Yaskawa INFORM job: A_ROOF_UPPER_0614_2_PAINT_9.JBI

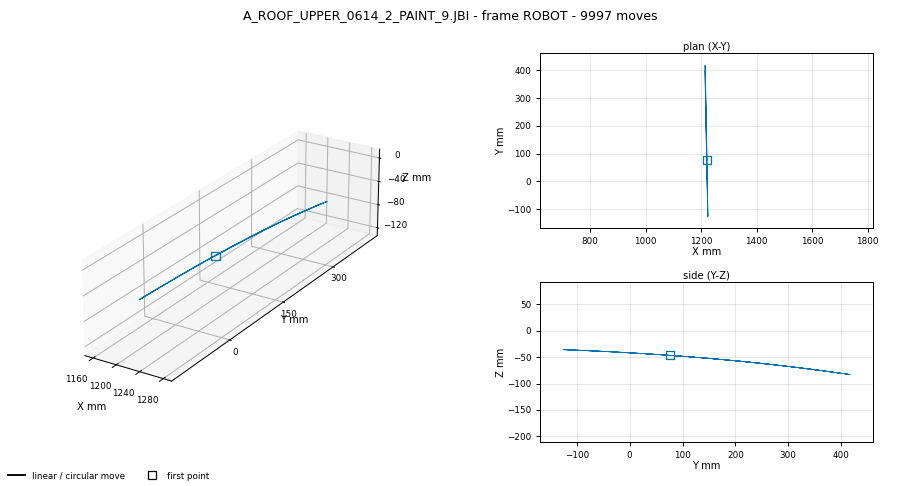
[picture p0: tool path of A_ROOF_UPPER_0614_2_PAINT_9.JBI in frame ROBOT, 9997 of 9997 moves have a stored position in this frame; points joined in program order, loops and branches not executed]
/JOB
//NAME A_ROOF_UPPER_0614_2_PAINT9
//POS
///NPOS 9997,0,0,0,0,0
///TOOL 1
///USER 0
///POSTYPE ROBOT
///RECTAN
///RCONF 1,0,0,0,0,0,0,0,0,0,0,0,0,0,0,0,0,0,0,0,0,0,0,0
C00000=1221.540,75.993,-46.507,-178.760,5.552,148.601
C00001=1221.535,76.242,-46.525,-178.757,5.552,148.601
C00002=1221.530,76.492,-46.542,-178.755,5.553,148.600
C00003=1221.525,76.741,-46.560,-178.753,5.554,148.600
C00004=1221.520,76.990,-46.578,-178.750,5.554,148.599
C00005=1221.515,77.240,-46.595,-178.747,5.555,148.598
C00006=1221.510,77.489,-46.613,-178.745,5.557,148.598
C00007=1221.505,77.738,-46.631,-178.742,5.557,148.597
C00008=1221.501,77.988,-46.648,-178.739,5.558,148.596
C00009=1221.496,78.237,-46.666,-178.737,5.559,148.596
C00010=1221.491,78.486,-46.684,-178.735,5.559,148.595
C00011=1221.486,78.735,-46.702,-178.732,5.560,148.595
C00012=1221.481,78.985,-46.719,-178.729,5.560,148.594
C00013=1221.476,79.234,-46.737,-178.727,5.561,148.594
C00014=1221.471,79.484,-46.755,-178.725,5.562,148.593
C00015=1221.466,79.733,-46.773,-178.722,5.563,148.592
C00016=1221.462,79.982,-46.790,-178.719,5.564,148.592
C00017=1221.457,80.231,-46.808,-178.717,5.565,148.591
C00018=1221.452,80.481,-46.826,-178.714,5.566,148.591
C00019=1221.448,80.730,-46.844,-178.711,5.566,148.590
C00020=1221.443,80.980,-46.862,-178.709,5.567,148.589
C00021=1221.437,81.249,-46.881,-178.707,5.568,148.589
C00022=1221.432,81.516,-46.900,-178.703,5.569,148.588
C00023=1221.427,81.784,-46.919,-178.701,5.570,148.588
C00024=1221.421,82.053,-46.939,-178.698,5.570,148.587
C00025=1221.416,82.302,-46.956,-178.696,5.571,148.586
C00026=1221.411,82.552,-46.974,-178.693,5.571,148.586
C00027=1221.407,82.801,-46.992,-178.690,5.573,148.585
C00028=1221.402,83.051,-47.010,-178.688,5.574,148.585
C00029=1221.397,83.300,-47.028,-178.685,5.574,148.584
C00030=1221.392,83.549,-47.046,-178.682,5.575,148.583
C00031=1221.387,83.798,-47.064,-178.680,5.576,148.583
C00032=1221.382,84.047,-47.082,-178.678,5.576,148.582
C00033=1221.378,84.296,-47.100,-178.675,5.577,148.581
C00034=1221.373,84.546,-47.118,-178.672,5.579,148.581
C00035=1221.368,84.796,-47.136,-178.670,5.579,148.580
C00036=1221.363,85.045,-47.154,-178.667,5.580,148.580
C00037=1221.358,85.294,-47.172,-178.664,5.581,148.579
C00038=1221.353,85.544,-47.190,-178.662,5.582,148.579
C00039=1221.348,85.793,-47.208,-178.660,5.582,148.578
C00040=1221.343,86.042,-47.226,-178.657,5.583,148.577
C00041=1221.339,86.291,-47.244,-178.654,5.584,148.577
C00042=1221.334,86.541,-47.262,-178.652,5.585,148.576
C00043=1221.329,86.790,-47.280,-178.649,5.586,148.576
C00044=1221.324,87.040,-47.298,-178.647,5.587,148.575
C00045=1221.319,87.289,-47.316,-178.644,5.587,148.575
C00046=1221.314,87.538,-47.334,-178.642,5.588,148.574
C00047=1221.309,87.787,-47.353,-178.639,5.588,148.573
C00048=1221.305,88.037,-47.371,-178.636,5.590,148.573
C00049=1221.300,88.286,-47.389,-178.634,5.591,148.572
C00050=1221.295,88.535,-47.407,-178.631,5.591,148.572
C00051=1221.290,88.784,-47.425,-178.629,5.592,148.571
C00052=1221.285,89.033,-47.443,-178.626,5.593,148.570
C00053=1221.281,89.283,-47.462,-178.624,5.593,148.570
C00054=1221.275,89.533,-47.480,-178.621,5.595,148.569
C00055=1221.270,89.782,-47.498,-178.618,5.596,148.569
C00056=1221.266,90.031,-47.516,-178.616,5.596,148.568
C00057=1221.261,90.279,-47.535,-178.614,5.597,148.568
C00058=1221.257,90.529,-47.553,-178.611,5.598,148.567
C00059=1221.252,90.779,-47.571,-178.608,5.599,148.566
C00060=1221.246,91.028,-47.590,-178.605,5.600,148.566
C00061=1221.241,91.277,-47.608,-178.603,5.601,148.565
C00062=1221.237,91.527,-47.626,-178.601,5.601,148.565
C00063=1221.232,91.776,-47.645,-178.598,5.602,148.564
C00064=1221.227,92.025,-47.663,-178.596,5.603,148.564
C00065=1221.222,92.274,-47.681,-178.593,5.604,148.563
C00066=1221.217,92.524,-47.700,-178.590,5.605,148.562
C00067=1221.212,92.773,-47.718,-178.588,5.606,148.562
C00068=1221.208,93.022,-47.736,-178.585,5.607,148.561
C00069=1221.203,93.271,-47.754,-178.583,5.607,148.561
C00070=1221.198,93.521,-47.773,-178.580,5.608,148.560
C00071=1221.193,93.770,-47.792,-178.577,5.610,148.560
C00072=1221.188,94.019,-47.810,-178.575,5.610,148.559
C00073=1221.183,94.268,-47.828,-178.573,5.611,148.558
C00074=1221.178,94.518,-47.847,-178.570,5.612,148.558
C00075=1221.174,94.767,-47.866,-178.567,5.612,148.557
C00076=1221.169,95.016,-47.884,-178.565,5.614,148.557
C00077=1221.165,95.266,-47.902,-178.562,5.615,148.556
C00078=1221.159,95.515,-47.921,-178.559,5.615,148.555
C00079=1221.154,95.764,-47.939,-178.557,5.616,148.555
C00080=1221.149,96.013,-47.957,-178.555,5.617,148.554
C00081=1221.145,96.263,-47.977,-178.551,5.618,148.554
C00082=1221.140,96.512,-47.995,-178.549,5.619,148.553
C00083=1221.135,96.761,-48.013,-178.547,5.620,148.553
C00084=1221.131,97.010,-48.032,-178.544,5.620,148.552
C00085=1221.125,97.260,-48.050,-178.542,5.621,148.552
C00086=1221.121,97.508,-48.069,-178.539,5.623,148.551
C00087=1221.116,97.758,-48.087,-178.537,5.624,148.551
C00088=1221.111,98.008,-48.106,-178.534,5.624,148.550
C00089=1221.106,98.256,-48.125,-178.531,5.625,148.549
C00090=1221.102,98.506,-48.143,-178.529,5.626,148.549
C00091=1221.096,98.755,-48.162,-178.526,5.627,148.548
C00092=1221.091,99.004,-48.180,-178.523,5.628,148.548
C00093=1221.087,99.254,-48.200,-178.521,5.629,148.547
C00094=1221.082,99.503,-48.218,-178.519,5.629,148.546
C00095=1221.078,99.752,-48.237,-178.516,5.631,148.546
C00096=1221.072,100.002,-48.256,-178.513,5.632,148.545
C00097=1221.068,100.250,-48.274,-178.511,5.632,148.545
C00098=1221.062,100.500,-48.293,-178.508,5.633,148.544
C00099=1221.058,100.749,-48.312,-178.506,5.634,148.544
C00100=1221.053,100.998,-48.330,-178.503,5.635,148.543
C00101=1221.048,101.248,-48.350,-178.501,5.636,148.543
C00102=1221.043,101.497,-48.368,-178.498,5.637,148.542
C00103=1221.039,101.747,-48.387,-178.496,5.638,148.541
C00104=1221.034,101.996,-48.405,-178.493,5.639,148.541
C00105=1221.028,102.245,-48.425,-178.490,5.640,148.540
C00106=1221.024,102.494,-48.444,-178.488,5.641,148.540
C00107=1221.019,102.743,-48.462,-178.485,5.641,148.539
C00108=1221.015,102.993,-48.481,-178.482,5.643,148.539
C00109=1221.010,103.242,-48.499,-178.480,5.644,148.538
C00110=1221.005,103.491,-48.519,-178.478,5.644,148.538
C00111=1221.000,103.740,-48.538,-178.475,5.645,148.537
C00112=1220.995,103.989,-48.556,-178.472,5.647,148.537
C00113=1220.991,104.239,-48.575,-178.470,5.647,148.536
C00114=1220.985,104.487,-48.594,-178.467,5.648,148.535
C00115=1220.981,104.737,-48.613,-178.465,5.649,148.535
C00116=1220.976,104.986,-48.632,-178.462,5.650,148.534
C00117=1220.972,105.235,-48.651,-178.460,5.651,148.534
C00118=1220.966,105.485,-48.670,-178.457,5.652,148.533
C00119=1220.961,105.735,-48.689,-178.454,5.653,148.532
C00120=1220.957,105.983,-48.708,-178.452,5.654,148.532
C00121=1220.952,106.233,-48.727,-178.449,5.655,148.531
C00122=1220.947,106.482,-48.746,-178.447,5.656,148.531
C00123=1220.942,106.731,-48.765,-178.444,5.657,148.530
C00124=1220.938,106.980,-48.784,-178.441,5.658,148.530
C00125=1220.932,107.249,-48.804,-178.439,5.659,148.529
C00126=1220.927,107.517,-48.825,-178.436,5.660,148.529
C00127=1220.921,107.785,-48.846,-178.433,5.661,148.528
C00128=1220.916,108.054,-48.866,-178.431,5.662,148.527
C00129=1220.912,108.303,-48.885,-178.428,5.663,148.527
C00130=1220.907,108.553,-48.905,-178.425,5.664,148.526
C00131=1220.903,108.802,-48.924,-178.423,5.665,148.526
C00132=1220.898,109.051,-48.943,-178.421,5.666,148.525
C00133=1220.892,109.301,-48.962,-178.417,5.667,148.525
C00134=1220.888,109.549,-48.981,-178.415,5.668,148.524
C00135=1220.883,109.799,-49.000,-178.413,5.669,148.524
C00136=1220.878,110.048,-49.020,-178.409,5.670,148.523
C00137=1220.874,110.297,-49.039,-178.407,5.671,148.523
C00138=1220.868,110.546,-49.058,-178.405,5.672,148.522
C00139=1220.864,110.796,-49.078,-178.403,5.673,148.522
C00140=1220.859,111.044,-49.096,-178.399,5.674,148.521
C00141=1220.854,111.294,-49.115,-178.397,5.675,148.520
C00142=1220.849,111.543,-49.134,-178.395,5.676,148.520
C00143=1220.845,111.792,-49.154,-178.392,5.677,148.519
C00144=1220.840,112.042,-49.173,-178.389,5.678,148.519
C00145=1220.835,112.291,-49.192,-178.387,5.679,148.518
C00146=1220.831,112.540,-49.212,-178.385,5.679,148.518
C00147=1220.825,112.789,-49.231,-178.381,5.681,148.517
C00148=1220.821,113.039,-49.250,-178.379,5.682,148.516
C00149=1220.815,113.287,-49.270,-178.377,5.682,148.516
C00150=1220.811,113.537,-49.289,-178.374,5.684,148.515
C00151=1220.806,113.786,-49.309,-178.371,5.685,148.515
C00152=1220.801,114.035,-49.328,-178.369,5.686,148.514
C00153=1220.796,114.285,-49.347,-178.367,5.686,148.514
C00154=1220.792,114.533,-49.366,-178.364,5.688,148.513
C00155=1220.787,114.783,-49.386,-178.361,5.689,148.513
C00156=1220.782,115.032,-49.405,-178.359,5.689,148.512
C00157=1220.777,115.281,-49.425,-178.356,5.691,148.512
C00158=1220.773,115.530,-49.444,-178.354,5.692,148.511
C00159=1220.768,115.780,-49.463,-178.351,5.692,148.511
C00160=1220.763,116.029,-49.483,-178.348,5.694,148.510
C00161=1220.758,116.278,-49.503,-178.346,5.695,148.510
C00162=1220.753,116.527,-49.522,-178.343,5.696,148.509
C00163=1220.748,116.776,-49.542,-178.340,5.697,148.509
C00164=1220.744,117.026,-49.561,-178.338,5.698,148.508
C00165=1220.739,117.274,-49.580,-178.336,5.699,148.507
C00166=1220.734,117.524,-49.600,-178.332,5.700,148.507
C00167=1220.729,117.774,-49.620,-178.330,5.701,148.506
C00168=1220.724,118.022,-49.639,-178.328,5.702,148.506
C00169=1220.720,118.271,-49.659,-178.325,5.704,148.505
C00170=1220.716,118.521,-49.678,-178.322,5.704,148.505
C00171=1220.710,118.769,-49.698,-178.320,5.705,148.504
C00172=1220.706,119.019,-49.717,-178.317,5.707,148.504
C00173=1220.701,119.269,-49.737,-178.315,5.708,148.503
C00174=1220.696,119.517,-49.757,-178.312,5.708,148.503
C00175=1220.691,119.766,-49.777,-178.309,5.710,148.502
C00176=1220.686,120.016,-49.796,-178.307,5.711,148.502
C00177=1220.682,120.266,-49.816,-178.304,5.711,148.501
C00178=1220.677,120.514,-49.836,-178.302,5.713,148.501
C00179=1220.672,120.763,-49.856,-178.299,5.714,148.500
C00180=1220.668,121.013,-49.875,-178.297,5.715,148.500
C00181=1220.662,121.261,-49.894,-178.294,5.716,148.499
C00182=1220.658,121.510,-49.914,-178.292,5.717,148.499
C00183=1220.653,121.760,-49.934,-178.289,5.718,148.498
C00184=1220.649,122.010,-49.954,-178.286,5.720,148.498
C00185=1220.643,122.258,-49.974,-178.284,5.720,148.497
C00186=1220.639,122.507,-49.993,-178.282,5.721,148.496
C00187=1220.634,122.757,-50.013,-178.279,5.723,148.496
C00188=1220.630,123.006,-50.033,-178.276,5.723,148.495
C00189=1220.624,123.255,-50.053,-178.274,5.724,148.495
C00190=1220.619,123.504,-50.072,-178.271,5.726,148.494
C00191=1220.615,123.753,-50.093,-178.269,5.727,148.494
C00192=1220.610,124.003,-50.112,-178.266,5.727,148.493
C00193=1220.605,124.251,-50.132,-178.263,5.729,148.493
C00194=1220.601,124.501,-50.152,-178.261,5.730,148.492
C00195=1220.596,124.750,-50.172,-178.258,5.731,148.492
C00196=1220.591,124.999,-50.192,-178.255,5.732,148.491
C00197=1220.586,125.248,-50.211,-178.253,5.733,148.491
C00198=1220.582,125.497,-50.232,-178.250,5.734,148.490
C00199=1220.577,125.747,-50.251,-178.248,5.735,148.490
C00200=1220.572,125.996,-50.272,-178.245,5.736,148.489
C00201=1220.568,126.245,-50.291,-178.243,5.738,148.489
C00202=1220.562,126.494,-50.312,-178.240,5.738,148.488
C00203=1220.557,126.743,-50.332,-178.238,5.739,148.488
C00204=1220.553,126.992,-50.352,-178.235,5.741,148.487
C00205=1220.548,127.242,-50.372,-178.233,5.742,148.487
C00206=1220.543,127.491,-50.392,-178.230,5.743,148.486
C00207=1220.539,127.740,-50.412,-178.227,5.744,148.486
C00208=1220.534,127.989,-50.432,-178.225,5.745,148.485
C00209=1220.529,128.238,-50.451,-178.222,5.747,148.485
C00210=1220.525,128.487,-50.472,-178.220,5.747,148.484
C00211=1220.520,128.737,-50.491,-178.217,5.749,148.484
C00212=1220.515,128.986,-50.512,-178.214,5.750,148.483
C00213=1220.510,129.235,-50.532,-178.212,5.751,148.482
C00214=1220.505,129.484,-50.552,-178.209,5.752,148.482
C00215=1220.500,129.733,-50.572,-178.207,5.753,148.481
C00216=1220.496,129.982,-50.592,-178.205,5.754,148.481
C00217=1220.491,130.231,-50.612,-178.202,5.755,148.480
C00218=1220.487,130.480,-50.633,-178.199,5.756,148.480
C00219=1220.481,130.730,-50.653,-178.196,5.758,148.479
C00220=1220.477,130.979,-50.673,-178.194,5.759,148.479
C00221=1220.472,131.228,-50.694,-178.192,5.759,148.478
C00222=1220.467,131.477,-50.713,-178.189,5.761,148.478
C00223=1220.463,131.726,-50.734,-178.186,5.762,148.477
C00224=1220.457,131.975,-50.754,-178.184,5.764,148.477
C00225=1220.453,132.225,-50.774,-178.181,5.764,148.476
C00226=1220.448,132.473,-50.794,-178.178,5.766,148.476
C00227=1220.444,132.722,-50.815,-178.176,5.767,148.475
C00228=1220.438,132.972,-50.835,-178.174,5.768,148.475
C00229=1220.434,133.240,-50.857,-178.170,5.769,148.474
C00230=1220.428,133.509,-50.879,-178.168,5.771,148.474
C00231=1220.423,133.778,-50.901,-178.165,5.772,148.473
C00232=1220.418,134.047,-50.922,-178.162,5.773,148.473
C00233=1220.413,134.296,-50.943,-178.160,5.774,148.472
C00234=1220.408,134.544,-50.963,-178.157,5.776,148.472
C00235=1220.404,134.793,-50.984,-178.155,5.776,148.471
C00236=1220.399,135.042,-51.004,-178.152,5.777,148.471
C00237=1220.394,135.292,-51.024,-178.149,5.779,148.470
C00238=1220.389,135.541,-51.045,-178.147,5.780,148.470
C00239=1220.385,135.790,-51.065,-178.144,5.781,148.469
C00240=1220.380,136.039,-51.086,-178.142,5.782,148.469
C00241=1220.375,136.288,-51.107,-178.139,5.784,148.468
C00242=1220.371,136.537,-51.127,-178.137,5.785,148.468
C00243=1220.366,136.787,-51.148,-178.134,5.785,148.467
C00244=1220.361,137.036,-51.167,-178.131,5.787,148.467
C00245=1220.357,137.285,-51.188,-178.129,5.788,148.466
C00246=1220.351,137.534,-51.209,-178.126,5.790,148.466
C00247=1220.347,137.783,-51.229,-178.124,5.791,148.465
C00248=1220.343,138.032,-51.250,-178.121,5.792,148.465
C00249=1220.337,138.282,-51.271,-178.119,5.793,148.464
C00250=1220.333,138.530,-51.291,-178.116,5.794,148.464
C00251=1220.328,138.780,-51.312,-178.113,5.795,148.463
C00252=1220.323,139.029,-51.332,-178.111,5.796,148.463
C00253=1220.319,139.278,-51.353,-178.108,5.798,148.462
C00254=1220.314,139.527,-51.374,-178.106,5.799,148.462
C00255=1220.309,139.776,-51.394,-178.103,5.800,148.461
C00256=1220.304,140.025,-51.415,-178.101,5.801,148.461
C00257=1220.300,140.274,-51.435,-178.098,5.803,148.460
C00258=1220.294,140.523,-51.456,-178.095,5.804,148.460
C00259=1220.290,140.772,-51.477,-178.092,5.805,148.459
C00260=1220.286,141.021,-51.497,-178.090,5.806,148.459
C00261=1220.280,141.270,-51.518,-178.088,5.808,148.459
C00262=1220.276,141.519,-51.538,-178.085,5.809,148.458
C00263=1220.271,141.769,-51.559,-178.083,5.810,148.458
C00264=1220.266,142.018,-51.580,-178.080,5.811,148.457
C00265=1220.262,142.268,-51.601,-178.078,5.812,148.457
C00266=1220.257,142.517,-51.621,-178.074,5.813,148.456
C00267=1220.252,142.766,-51.642,-178.072,5.814,148.456
C00268=1220.248,143.014,-51.663,-178.070,5.816,148.455
C00269=1220.243,143.263,-51.684,-178.067,5.817,148.454
C00270=1220.238,143.512,-51.705,-178.064,5.819,148.454
C00271=1220.233,143.762,-51.726,-178.062,5.819,148.453
C00272=1220.229,144.011,-51.746,-178.059,5.821,148.453
C00273=1220.224,144.260,-51.767,-178.057,5.822,148.453
C00274=1220.220,144.508,-51.788,-178.054,5.824,148.452
C00275=1220.215,144.758,-51.810,-178.052,5.825,148.452
C00276=1220.210,145.007,-51.830,-178.049,5.826,148.451
C00277=1220.205,145.256,-51.851,-178.046,5.827,148.451
C00278=1220.200,145.506,-51.872,-178.044,5.829,148.450
C00279=1220.196,145.754,-51.893,-178.041,5.829,148.450
C00280=1220.191,146.003,-51.914,-178.039,5.831,148.449
C00281=1220.186,146.252,-51.934,-178.036,5.832,148.449
C00282=1220.181,146.501,-51.955,-178.033,5.834,148.448
C00283=1220.177,146.751,-51.977,-178.031,5.835,148.448
C00284=1220.173,147.000,-51.998,-178.028,5.836,148.447
C00285=1220.167,147.249,-52.019,-178.026,5.837,148.447
C00286=1220.162,147.498,-52.040,-178.023,5.839,148.447
C00287=1220.158,147.746,-52.061,-178.021,5.840,148.446
C00288=1220.153,147.996,-52.082,-178.018,5.841,148.446
C00289=1220.148,148.245,-52.102,-178.015,5.842,148.445
C00290=1220.144,148.494,-52.124,-178.013,5.844,148.445
C00291=1220.139,148.743,-52.145,-178.011,5.845,148.444
C00292=1220.135,148.992,-52.165,-178.007,5.846,148.444
C00293=1220.130,149.241,-52.187,-178.005,5.847,148.443
C00294=1220.125,149.490,-52.208,-178.003,5.849,148.443
C00295=1220.121,149.740,-52.229,-178.000,5.850,148.442
C00296=1220.116,149.988,-52.250,-177.997,5.852,148.442
C00297=1220.111,150.238,-52.271,-177.995,5.852,148.441
C00298=1220.106,150.486,-52.293,-177.992,5.854,148.441
C00299=1220.101,150.735,-52.313,-177.990,5.855,148.440
C00300=1220.097,150.985,-52.336,-177.987,5.856,148.440
C00301=1220.092,151.234,-52.356,-177.985,5.857,148.439
C00302=1220.087,151.483,-52.377,-177.982,5.859,148.439
C00303=1220.083,151.731,-52.399,-177.979,5.860,148.438
C00304=1220.078,151.981,-52.420,-177.977,5.862,148.438
C00305=1220.073,152.230,-52.442,-177.975,5.863,148.438
C00306=1220.069,152.479,-52.462,-177.972,5.864,148.437
C00307=1220.064,152.728,-52.484,-177.969,5.866,148.437
C00308=1220.059,152.977,-52.505,-177.967,5.867,148.436
C00309=1220.054,153.226,-52.527,-177.964,5.868,148.436
C00310=1220.049,153.476,-52.548,-177.962,5.869,148.435
C00311=1220.045,153.724,-52.569,-177.958,5.871,148.435
C00312=1220.040,153.973,-52.590,-177.956,5.872,148.434
C00313=1220.036,154.222,-52.612,-177.954,5.874,148.434
C00314=1220.031,154.471,-52.633,-177.951,5.874,148.433
C00315=1220.026,154.720,-52.654,-177.948,5.876,148.433
C00316=1220.022,154.969,-52.676,-177.946,5.877,148.433
C00317=1220.017,155.219,-52.697,-177.943,5.879,148.432
C00318=1220.012,155.467,-52.718,-177.941,5.880,148.432
C00319=1220.007,155.716,-52.740,-177.938,5.881,148.431
C00320=1220.003,155.966,-52.761,-177.935,5.883,148.431
C00321=1219.998,156.215,-52.783,-177.933,5.884,148.430
C00322=1219.993,156.464,-52.804,-177.930,5.886,148.430
C00323=1219.989,156.713,-52.826,-177.928,5.886,148.429
C00324=1219.984,156.961,-52.847,-177.925,5.888,148.429
C00325=1219.979,157.211,-52.868,-177.923,5.889,148.428
C00326=1219.975,157.460,-52.890,-177.920,5.891,148.428
C00327=1219.970,157.709,-52.912,-177.917,5.892,148.427
C00328=1219.965,157.957,-52.934,-177.915,5.893,148.427
C00329=1219.960,158.207,-52.955,-177.912,5.895,148.427
C00330=1219.956,158.456,-52.977,-177.910,5.896,148.426
C00331=1219.951,158.705,-52.998,-177.907,5.898,148.426
C00332=1219.946,158.955,-53.020,-177.905,5.899,148.425
C00333=1219.942,159.223,-53.043,-177.902,5.900,148.425
C00334=1219.936,159.492,-53.066,-177.899,5.902,148.424
C00335=1219.931,159.761,-53.089,-177.896,5.903,148.424
C00336=1219.926,160.030,-53.113,-177.894,5.904,148.423
C00337=1219.921,160.279,-53.135,-177.891,5.906,148.423
C00338=1219.917,160.529,-53.156,-177.888,5.908,148.422
C00339=1219.912,160.777,-53.178,-177.886,5.909,148.422
C00340=1219.907,161.026,-53.200,-177.883,5.910,148.421
C00341=1219.903,161.275,-53.222,-177.881,5.911,148.421
C00342=1219.898,161.524,-53.243,-177.878,5.913,148.421
C00343=1219.893,161.773,-53.265,-177.876,5.915,148.420
C00344=1219.888,162.023,-53.286,-177.873,5.915,148.420
C00345=1219.884,162.271,-53.308,-177.870,5.917,148.419
C00346=1219.879,162.521,-53.330,-177.868,5.918,148.419
C00347=1219.874,162.769,-53.352,-177.865,5.920,148.418
C00348=1219.870,163.019,-53.374,-177.862,5.922,148.418
C00349=1219.865,163.267,-53.396,-177.860,5.923,148.418
C00350=1219.860,163.516,-53.417,-177.857,5.924,148.417
C00351=1219.856,163.765,-53.439,-177.855,5.925,148.417
C00352=1219.851,164.014,-53.461,-177.852,5.927,148.416
C00353=1219.847,164.263,-53.483,-177.850,5.929,148.416
C00354=1219.841,164.512,-53.505,-177.847,5.929,148.415
C00355=1219.837,164.761,-53.527,-177.844,5.931,148.415
C00356=1219.832,165.010,-53.549,-177.842,5.932,148.414
C00357=1219.828,165.259,-53.571,-177.840,5.934,148.414
C00358=1219.823,165.508,-53.593,-177.837,5.935,148.414
C00359=1219.818,165.757,-53.614,-177.834,5.936,148.413
C00360=1219.814,166.006,-53.637,-177.832,5.938,148.413
C00361=1219.809,166.255,-53.658,-177.829,5.939,148.412
C00362=1219.805,166.504,-53.680,-177.827,5.941,148.412
C00363=1219.799,166.753,-53.703,-177.824,5.942,148.411
C00364=1219.795,167.002,-53.725,-177.822,5.943,148.411
C00365=1219.790,167.251,-53.746,-177.819,5.945,148.410
C00366=1219.786,167.500,-53.768,-177.816,5.947,148.410
C00367=1219.781,167.749,-53.790,-177.814,5.948,148.410
C00368=1219.777,167.998,-53.812,-177.811,5.950,148.409
C00369=1219.771,168.247,-53.835,-177.809,5.950,148.409
C00370=1219.767,168.496,-53.857,-177.806,5.952,148.408
C00371=1219.762,168.745,-53.879,-177.803,5.954,148.408
C00372=1219.758,168.994,-53.901,-177.801,5.955,148.408
C00373=1219.753,169.243,-53.923,-177.798,5.956,148.407
C00374=1219.748,169.492,-53.945,-177.795,5.958,148.407
C00375=1219.744,169.742,-53.967,-177.793,5.959,148.406
C00376=1219.739,169.990,-53.990,-177.791,5.961,148.406
C00377=1219.735,170.239,-54.012,-177.787,5.963,148.405
C00378=1219.729,170.488,-54.034,-177.785,5.963,148.405
C00379=1219.725,170.737,-54.056,-177.783,5.965,148.405
C00380=1219.721,170.985,-54.078,-177.780,5.967,148.404
C00381=1219.716,171.235,-54.100,-177.778,5.968,148.404
C00382=1219.711,171.484,-54.123,-177.775,5.970,148.403
C00383=1219.706,171.733,-54.145,-177.773,5.971,148.403
C00384=1219.703,171.982,-54.168,-177.770,5.972,148.402
C00385=1219.697,172.231,-54.190,-177.767,5.974,148.402
C00386=1219.693,172.480,-54.212,-177.765,5.975,148.402
C00387=1219.688,172.729,-54.234,-177.762,5.977,148.401
C00388=1219.683,172.978,-54.257,-177.760,5.979,148.401
C00389=1219.678,173.226,-54.279,-177.757,5.980,148.400
C00390=1219.674,173.476,-54.301,-177.754,5.981,148.400
C00391=1219.669,173.725,-54.324,-177.752,5.983,148.399
C00392=1219.664,173.973,-54.346,-177.750,5.984,148.399
C00393=1219.660,174.223,-54.368,-177.747,5.986,148.399
C00394=1219.655,174.472,-54.391,-177.744,5.987,148.398
C00395=1219.651,174.720,-54.413,-177.742,5.988,148.398
C00396=1219.647,174.969,-54.436,-177.739,5.990,148.397
C00397=1219.641,175.218,-54.458,-177.736,5.992,148.397
C00398=1219.637,175.467,-54.480,-177.734,5.993,148.397
C00399=1219.632,175.716,-54.503,-177.731,5.994,148.396
C00400=1219.627,175.965,-54.525,-177.728,5.996,148.396
C00401=1219.623,176.214,-54.548,-177.726,5.998,148.395
C00402=1219.618,176.463,-54.570,-177.724,5.999,148.395
C00403=1219.614,176.711,-54.593,-177.721,6.001,148.395
C00404=1219.609,176.961,-54.615,-177.718,6.002,148.394
C00405=1219.605,177.210,-54.638,-177.716,6.003,148.394
C00406=1219.600,177.458,-54.660,-177.713,6.005,148.393
C00407=1219.595,177.707,-54.683,-177.711,6.007,148.393
C00408=1219.591,177.957,-54.705,-177.708,6.008,148.393
C00409=1219.586,178.205,-54.728,-177.705,6.009,148.392
C00410=1219.581,178.454,-54.750,-177.703,6.011,148.392
C00411=1219.577,178.703,-54.774,-177.701,6.012,148.391
C00412=1219.572,178.952,-54.795,-177.698,6.014,148.391
C00413=1219.567,179.201,-54.819,-177.695,6.016,148.391
C00414=1219.563,179.450,-54.841,-177.692,6.017,148.390
C00415=1219.557,179.699,-54.864,-177.690,6.018,148.390
C00416=1219.553,179.947,-54.886,-177.687,6.020,148.389
C00417=1219.548,180.197,-54.909,-177.685,6.022,148.389
C00418=1219.544,180.446,-54.932,-177.683,6.023,148.388
C00419=1219.539,180.694,-54.955,-177.679,6.025,148.388
C00420=1219.535,180.944,-54.977,-177.677,6.026,148.388
C00421=1219.530,181.193,-55.000,-177.674,6.028,148.387
C00422=1219.525,181.442,-55.024,-177.672,6.029,148.387
C00423=1219.521,181.690,-55.045,-177.669,6.031,148.386
C00424=1219.516,181.939,-55.069,-177.667,6.033,148.386
C00425=1219.512,182.188,-55.091,-177.664,6.034,148.385
C00426=1219.507,182.438,-55.114,-177.662,6.035,148.385
C00427=1219.502,182.686,-55.136,-177.659,6.037,148.385
C00428=1219.498,182.935,-55.160,-177.656,6.039,148.384
C00429=1219.493,183.184,-55.183,-177.654,6.040,148.384
C00430=1219.489,183.433,-55.205,-177.651,6.042,148.384
C00431=1219.483,183.681,-55.228,-177.648,6.043,148.383
C00432=1219.479,183.930,-55.251,-177.646,6.044,148.383
C00433=1219.475,184.179,-55.274,-177.644,6.046,148.382
C00434=1219.470,184.429,-55.297,-177.641,6.048,148.382
C00435=1219.466,184.678,-55.320,-177.638,6.050,148.382
C00436=1219.460,184.926,-55.343,-177.636,6.051,148.381
C00437=1219.455,185.196,-55.368,-177.633,6.052,148.381
C00438=1219.451,185.465,-55.392,-177.630,6.054,148.380
C00439=1219.446,185.736,-55.418,-177.628,6.056,148.380
C00440=1219.441,186.005,-55.443,-177.625,6.058,148.379
C00441=1219.436,186.253,-55.465,-177.622,6.059,148.379
C00442=1219.431,186.502,-55.488,-177.619,6.061,148.379
C00443=1219.427,186.751,-55.512,-177.617,6.063,148.378
C00444=1219.423,187.000,-55.535,-177.615,6.064,148.378
C00445=1219.418,187.249,-55.558,-177.612,6.066,148.378
C00446=1219.413,187.498,-55.581,-177.609,6.067,148.377
C00447=1219.409,187.746,-55.604,-177.606,6.069,148.377
C00448=1219.404,187.996,-55.626,-177.604,6.070,148.376
C00449=1219.399,188.245,-55.650,-177.601,6.072,148.376
C00450=1219.394,188.494,-55.673,-177.599,6.074,148.376
C00451=1219.390,188.743,-55.696,-177.596,6.076,148.375
C00452=1219.386,188.992,-55.719,-177.594,6.077,148.375
C00453=1219.381,189.241,-55.742,-177.591,6.079,148.375
C00454=1219.376,189.490,-55.766,-177.588,6.080,148.374
C00455=1219.371,189.738,-55.789,-177.586,6.082,148.374
C00456=1219.367,189.987,-55.812,-177.584,6.083,148.373
C00457=1219.362,190.236,-55.835,-177.581,6.085,148.373
C00458=1219.358,190.485,-55.858,-177.578,6.087,148.373
C00459=1219.353,190.734,-55.882,-177.576,6.088,148.372
C00460=1219.348,190.982,-55.906,-177.573,6.090,148.372
C00461=1219.344,191.231,-55.929,-177.571,6.091,148.372
C00462=1219.340,191.480,-55.952,-177.568,6.093,148.371
C00463=1219.335,191.729,-55.975,-177.565,6.095,148.371
C00464=1219.330,191.978,-55.999,-177.562,6.096,148.370
C00465=1219.325,192.226,-56.022,-177.560,6.098,148.370
C00466=1219.320,192.475,-56.045,-177.558,6.099,148.370
C00467=1219.316,192.724,-56.068,-177.555,6.101,148.369
C00468=1219.311,192.974,-56.092,-177.552,6.103,148.369
C00469=1219.307,193.222,-56.115,-177.550,6.105,148.368
C00470=1219.303,193.471,-56.138,-177.548,6.106,148.368
C00471=1219.298,193.720,-56.162,-177.545,6.108,148.368
C00472=1219.293,193.969,-56.185,-177.542,6.109,148.367
C00473=1219.289,194.218,-56.209,-177.539,6.111,148.367
C00474=1219.284,194.466,-56.233,-177.537,6.113,148.366
C00475=1219.279,194.715,-56.256,-177.534,6.114,148.366
C00476=1219.275,194.964,-56.279,-177.532,6.116,148.366
C00477=1219.270,195.213,-56.303,-177.529,6.117,148.365
C00478=1219.265,195.462,-56.326,-177.527,6.119,148.365
C00479=1219.261,195.711,-56.350,-177.524,6.121,148.365
C00480=1219.256,195.960,-56.373,-177.521,6.123,148.364
C00481=1219.252,196.209,-56.397,-177.519,6.124,148.364
C00482=1219.247,196.457,-56.421,-177.517,6.126,148.364
C00483=1219.242,196.706,-56.444,-177.514,6.128,148.363
C00484=1219.238,196.955,-56.468,-177.511,6.129,148.363
C00485=1219.233,197.204,-56.492,-177.508,6.131,148.362
C00486=1219.229,197.453,-56.515,-177.506,6.132,148.362
C00487=1219.224,197.702,-56.538,-177.503,6.134,148.362
C00488=1219.220,197.950,-56.563,-177.501,6.136,148.361
C00489=1219.215,198.199,-56.586,-177.498,6.138,148.361
C00490=1219.210,198.448,-56.609,-177.495,6.139,148.361
C00491=1219.206,198.697,-56.633,-177.493,6.141,148.360
C00492=1219.201,198.946,-56.657,-177.491,6.142,148.360
C00493=1219.197,199.194,-56.681,-177.488,6.144,148.360
C00494=1219.192,199.443,-56.704,-177.485,6.146,148.359
C00495=1219.187,199.692,-56.727,-177.483,6.148,148.359
C00496=1219.183,199.941,-56.752,-177.480,6.150,148.359
C00497=1219.178,200.190,-56.775,-177.478,6.151,148.358
C00498=1219.174,200.439,-56.799,-177.475,6.152,148.358
C00499=1219.170,200.688,-56.823,-177.472,6.154,148.357
C00500=1219.165,200.936,-56.847,-177.470,6.156,148.357
C00501=1219.160,201.185,-56.871,-177.467,6.158,148.357
C00502=1219.155,201.434,-56.895,-177.464,6.159,148.356
C00503=1219.151,201.683,-56.918,-177.462,6.161,148.356
C00504=1219.146,201.931,-56.942,-177.460,6.162,148.356
C00505=1219.142,202.180,-56.966,-177.457,6.164,148.355
C00506=1219.137,202.429,-56.990,-177.454,6.166,148.355
C00507=1219.133,202.678,-57.013,-177.452,6.168,148.355
C00508=1219.128,202.927,-57.038,-177.449,6.170,148.354
C00509=1219.124,203.176,-57.062,-177.446,6.172,148.354
C00510=1219.119,203.425,-57.085,-177.444,6.173,148.354
C00511=1219.115,203.673,-57.110,-177.441,6.175,148.353
C00512=1219.110,203.922,-57.133,-177.439,6.176,148.353
C00513=1219.105,204.171,-57.158,-177.436,6.178,148.352
C00514=1219.100,204.419,-57.182,-177.434,6.180,148.352
C00515=1219.096,204.669,-57.205,-177.431,6.182,148.352
C00516=1219.092,204.917,-57.229,-177.429,6.184,148.351
C00517=1219.087,205.166,-57.254,-177.426,6.185,148.351
C00518=1219.082,205.415,-57.277,-177.423,6.187,148.351
C00519=1219.078,205.664,-57.302,-177.421,6.188,148.350
C00520=1219.073,205.912,-57.326,-177.419,6.190,148.350
C00521=1219.069,206.162,-57.349,-177.416,6.192,148.350
C00522=1219.064,206.410,-57.374,-177.413,6.194,148.349
C00523=1219.060,206.659,-57.398,-177.411,6.196,148.349
C00524=1219.055,206.907,-57.422,-177.408,6.198,148.349
C00525=1219.051,207.156,-57.446,-177.405,6.199,148.348
C00526=1219.045,207.405,-57.470,-177.403,6.201,148.348
C00527=1219.042,207.654,-57.495,-177.400,6.203,148.348
C00528=1219.037,207.903,-57.519,-177.398,6.204,148.347
C00529=1219.032,208.152,-57.543,-177.395,6.206,148.347
C00530=1219.027,208.400,-57.567,-177.393,6.208,148.347
C00531=1219.024,208.649,-57.591,-177.390,6.210,148.346
C00532=1219.018,208.898,-57.616,-177.387,6.211,148.346
C00533=1219.014,209.147,-57.640,-177.385,6.213,148.346
C00534=1219.010,209.395,-57.664,-177.382,6.215,148.345
C00535=1219.004,209.644,-57.688,-177.380,6.217,148.345
C00536=1219.000,209.893,-57.712,-177.377,6.219,148.345
C00537=1218.995,210.142,-57.737,-177.374,6.221,148.344
C00538=1218.991,210.391,-57.761,-177.372,6.222,148.344
C00539=1218.986,210.639,-57.785,-177.370,6.224,148.344
C00540=1218.982,210.888,-57.810,-177.367,6.225,148.343
C00541=1218.977,211.159,-57.837,-177.364,6.227,148.343
C00542=1218.972,211.429,-57.862,-177.361,6.230,148.342
C00543=1218.967,211.699,-57.889,-177.358,6.231,148.342
C00544=1218.962,211.970,-57.916,-177.355,6.233,148.342
C00545=1218.958,212.218,-57.940,-177.353,6.235,148.341
C00546=1218.953,212.467,-57.965,-177.350,6.237,148.341
C00547=1218.948,212.716,-57.989,-177.347,6.239,148.341
C00548=1218.944,212.965,-58.014,-177.345,6.241,148.340
C00549=1218.940,213.213,-58.038,-177.342,6.243,148.340
C00550=1218.934,213.462,-58.063,-177.340,6.244,148.340
C00551=1218.931,213.711,-58.087,-177.337,6.245,148.339
C00552=1218.925,213.960,-58.112,-177.335,6.247,148.339
C00553=1218.921,214.208,-58.136,-177.332,6.249,148.339
C00554=1218.917,214.458,-58.161,-177.330,6.251,148.338
C00555=1218.912,214.706,-58.185,-177.327,6.253,148.338
C00556=1218.907,214.955,-58.210,-177.324,6.255,148.338
C00557=1218.903,215.204,-58.234,-177.322,6.257,148.337
C00558=1218.898,215.452,-58.260,-177.319,6.258,148.337
C00559=1218.894,215.701,-58.284,-177.317,6.261,148.337
C00560=1218.889,215.950,-58.309,-177.314,6.262,148.337
C00561=1218.885,216.198,-58.333,-177.312,6.264,148.336
C00562=1218.880,216.447,-58.357,-177.309,6.266,148.336
C00563=1218.876,216.696,-58.382,-177.306,6.268,148.336
C00564=1218.871,216.944,-58.407,-177.304,6.270,148.335
C00565=1218.866,217.193,-58.432,-177.301,6.272,148.335
C00566=1218.862,217.442,-58.456,-177.298,6.274,148.335
C00567=1218.857,217.691,-58.481,-177.296,6.275,148.334
C00568=1218.853,217.940,-58.505,-177.294,6.276,148.334
C00569=1218.849,218.188,-58.531,-177.291,6.278,148.334
C00570=1218.844,218.437,-58.556,-177.288,6.280,148.333
C00571=1218.840,218.686,-58.580,-177.286,6.282,148.333
C00572=1218.835,218.935,-58.605,-177.283,6.284,148.333
C00573=1218.831,219.183,-58.630,-177.281,6.286,148.332
C00574=1218.826,219.432,-58.654,-177.278,6.287,148.332
C00575=1218.821,219.681,-58.679,-177.275,6.289,148.332
C00576=1218.817,219.929,-58.704,-177.273,6.292,148.332
C00577=1218.812,220.178,-58.729,-177.270,6.293,148.331
C00578=1218.808,220.427,-58.754,-177.268,6.295,148.331
C00579=1218.804,220.675,-58.779,-177.265,6.297,148.331
C00580=1218.799,220.925,-58.804,-177.263,6.299,148.330
C00581=1218.794,221.173,-58.828,-177.260,6.301,148.330
C00582=1218.790,221.422,-58.854,-177.257,6.303,148.330
C00583=1218.785,221.670,-58.878,-177.255,6.305,148.329
C00584=1218.781,221.920,-58.903,-177.252,6.306,148.329
C00585=1218.776,222.168,-58.929,-177.249,6.308,148.329
C00586=1218.772,222.416,-58.953,-177.247,6.310,148.328
C00587=1218.767,222.665,-58.979,-177.245,6.312,148.328
C00588=1218.762,222.914,-59.003,-177.242,6.314,148.328
C00589=1218.758,223.163,-59.029,-177.239,6.316,148.327
C00590=1218.754,223.411,-59.053,-177.237,6.318,148.327
C00591=1218.749,223.660,-59.079,-177.234,6.320,148.327
C00592=1218.744,223.909,-59.103,-177.231,6.322,148.326
C00593=1218.740,224.158,-59.129,-177.229,6.323,148.326
C00594=1218.736,224.406,-59.153,-177.226,6.325,148.326
C00595=1218.731,224.655,-59.179,-177.224,6.327,148.326
C00596=1218.726,224.903,-59.204,-177.221,6.329,148.325
C00597=1218.722,225.152,-59.229,-177.219,6.331,148.325
C00598=1218.717,225.401,-59.254,-177.216,6.333,148.325
C00599=1218.713,225.650,-59.280,-177.214,6.335,148.324
C00600=1218.708,225.898,-59.304,-177.211,6.337,148.324
C00601=1218.704,226.147,-59.330,-177.209,6.338,148.324
C00602=1218.700,226.396,-59.355,-177.206,6.340,148.323
C00603=1218.695,226.645,-59.380,-177.204,6.341,148.323
C00604=1218.690,226.893,-59.406,-177.201,6.344,148.323
C00605=1218.685,227.142,-59.431,-177.199,6.345,148.323
C00606=1218.681,227.391,-59.456,-177.196,6.347,148.322
C00607=1218.677,227.639,-59.481,-177.194,6.349,148.322
C00608=1218.673,227.888,-59.506,-177.191,6.351,148.322
C00609=1218.668,228.136,-59.531,-177.188,6.353,148.321
C00610=1218.663,228.385,-59.557,-177.186,6.355,148.321
C00611=1218.659,228.634,-59.582,-177.184,6.357,148.321
C00612=1218.654,228.883,-59.608,-177.181,6.359,148.321
C00613=1218.650,229.131,-59.633,-177.178,6.361,148.320
C00614=1218.645,229.379,-59.659,-177.176,6.363,148.320
C00615=1218.641,229.629,-59.684,-177.173,6.364,148.320
C00616=1218.636,229.878,-59.710,-177.170,6.366,148.319
C00617=1218.631,230.126,-59.735,-177.168,6.368,148.319
C00618=1218.627,230.375,-59.761,-177.166,6.370,148.319
C00619=1218.622,230.623,-59.785,-177.163,6.372,148.319
C00620=1218.618,230.872,-59.811,-177.160,6.374,148.318
C00621=1218.614,231.121,-59.837,-177.158,6.376,148.318
C00622=1218.609,231.369,-59.862,-177.155,6.379,148.318
C00623=1218.605,231.618,-59.888,-177.152,6.380,148.317
C00624=1218.600,231.867,-59.913,-177.150,6.383,148.317
C00625=1218.595,232.115,-59.938,-177.147,6.384,148.317
C00626=1218.591,232.364,-59.964,-177.145,6.386,148.317
C00627=1218.587,232.613,-59.990,-177.142,6.388,148.316
C00628=1218.582,232.861,-60.015,-177.139,6.390,148.316
C00629=1218.578,233.110,-60.041,-177.137,6.392,148.316
C00630=1218.574,233.359,-60.067,-177.135,6.394,148.316
C00631=1218.569,233.607,-60.092,-177.132,6.396,148.315
C00632=1218.564,233.856,-60.118,-177.129,6.398,148.315
C00633=1218.560,234.105,-60.143,-177.127,6.400,148.315
C00634=1218.555,234.353,-60.168,-177.125,6.402,148.314
C00635=1218.551,234.602,-60.194,-177.122,6.404,148.314
C00636=1218.547,234.851,-60.220,-177.119,6.406,148.314
C00637=1218.542,235.099,-60.245,-177.117,6.407,148.314
C00638=1218.537,235.348,-60.272,-177.114,6.409,148.313
C00639=1218.533,235.597,-60.297,-177.112,6.411,148.313
C00640=1218.528,235.845,-60.323,-177.109,6.413,148.313
C00641=1218.524,236.094,-60.349,-177.107,6.415,148.312
C00642=1218.519,236.342,-60.374,-177.104,6.417,148.312
C00643=1218.515,236.591,-60.400,-177.101,6.419,148.312
C00644=1218.511,236.839,-60.426,-177.099,6.421,148.312
C00645=1218.506,237.111,-60.454,-177.097,6.423,148.311
C00646=1218.501,237.383,-60.483,-177.093,6.426,148.311
C00647=1218.496,237.653,-60.511,-177.091,6.428,148.311
C00648=1218.491,237.925,-60.539,-177.088,6.429,148.310
C00649=1218.486,238.173,-60.565,-177.086,6.431,148.310
C00650=1218.482,238.422,-60.590,-177.082,6.434,148.310
C00651=1218.478,238.671,-60.616,-177.080,6.436,148.310
C00652=1218.473,238.920,-60.642,-177.078,6.438,148.309
C00653=1218.469,239.168,-60.669,-177.075,6.440,148.309
C00654=1218.464,239.416,-60.694,-177.072,6.442,148.309
C00655=1218.460,239.665,-60.720,-177.070,6.444,148.309
C00656=1218.455,239.914,-60.746,-177.068,6.446,148.308
C00657=1218.450,240.163,-60.772,-177.065,6.448,148.308
C00658=1218.446,240.411,-60.798,-177.062,6.450,148.308
C00659=1218.442,240.659,-60.824,-177.060,6.451,148.307
C00660=1218.437,240.909,-60.850,-177.058,6.454,148.307
C00661=1218.433,241.157,-60.876,-177.055,6.455,148.307
C00662=1218.429,241.406,-60.903,-177.052,6.457,148.307
C00663=1218.424,241.654,-60.928,-177.050,6.459,148.306
C00664=1218.419,241.903,-60.954,-177.048,6.461,148.306
C00665=1218.415,242.152,-60.980,-177.045,6.463,148.306
C00666=1218.411,242.400,-61.007,-177.042,6.466,148.306
C00667=1218.406,242.649,-61.033,-177.040,6.468,148.306
C00668=1218.401,242.898,-61.059,-177.037,6.470,148.305
C00669=1218.397,243.145,-61.085,-177.034,6.472,148.305
C00670=1218.392,243.394,-61.111,-177.032,6.474,148.305
C00671=1218.388,243.642,-61.138,-177.030,6.476,148.305
C00672=1218.384,243.891,-61.163,-177.027,6.478,148.304
C00673=1218.379,244.140,-61.190,-177.024,6.480,148.304
C00674=1218.375,244.389,-61.216,-177.022,6.481,148.304
C00675=1218.370,244.638,-61.242,-177.020,6.484,148.304
C00676=1218.366,244.886,-61.269,-177.017,6.486,148.303
C00677=1218.361,245.134,-61.294,-177.014,6.487,148.303
C00678=1218.356,245.383,-61.321,-177.012,6.490,148.303
C00679=1218.352,245.631,-61.347,-177.009,6.492,148.303
C00680=1218.347,245.880,-61.373,-177.007,6.494,148.302
C00681=1218.344,246.129,-61.400,-177.004,6.496,148.302
C00682=1218.339,246.378,-61.426,-177.002,6.498,148.302
C00683=1218.335,246.626,-61.453,-176.999,6.500,148.302
C00684=1218.330,246.875,-61.478,-176.997,6.502,148.301
C00685=1218.326,247.123,-61.506,-176.994,6.504,148.301
C00686=1218.322,247.372,-61.531,-176.992,6.506,148.301
C00687=1218.316,247.620,-61.558,-176.989,6.508,148.301
C00688=1218.312,247.869,-61.584,-176.986,6.511,148.301
C00689=1218.307,248.117,-61.611,-176.984,6.513,148.300
C00690=1218.303,248.365,-61.637,-176.981,6.515,148.300
C00691=1218.299,248.614,-61.664,-176.979,6.517,148.300
C00692=1218.295,248.863,-61.690,-176.976,6.519,148.300
C00693=1218.290,249.112,-61.716,-176.974,6.521,148.299
C00694=1218.286,249.360,-61.743,-176.971,6.522,148.299
C00695=1218.281,249.608,-61.770,-176.969,6.525,148.299
C00696=1218.276,249.857,-61.796,-176.967,6.527,148.298
C00697=1218.272,250.106,-61.823,-176.963,6.529,148.298
C00698=1218.268,250.354,-61.850,-176.961,6.531,148.298
C00699=1218.263,250.603,-61.876,-176.959,6.533,148.298
C00700=1218.259,250.851,-61.903,-176.956,6.535,148.298
C00701=1218.255,251.100,-61.929,-176.954,6.537,148.297
C00702=1218.250,251.349,-61.955,-176.951,6.539,148.297
C00703=1218.245,251.597,-61.982,-176.949,6.541,148.297
C00704=1218.241,251.845,-62.009,-176.946,6.544,148.297
C00705=1218.237,252.094,-62.036,-176.943,6.546,148.296
C00706=1218.232,252.343,-62.062,-176.941,6.548,148.296
C00707=1218.228,252.591,-62.089,-176.939,6.550,148.296
C00708=1218.223,252.840,-62.116,-176.936,6.552,148.296
C00709=1218.219,253.088,-62.142,-176.933,6.554,148.295
C00710=1218.214,253.336,-62.169,-176.931,6.556,148.295
C00711=1218.209,253.586,-62.196,-176.929,6.558,148.295
C00712=1218.206,253.834,-62.222,-176.926,6.561,148.295
C00713=1218.201,254.082,-62.249,-176.923,6.563,148.295
C00714=1218.196,254.331,-62.276,-176.921,6.565,148.294
C00715=1218.192,254.579,-62.303,-176.919,6.567,148.294
C00716=1218.188,254.827,-62.330,-176.916,6.569,148.294
C00717=1218.183,255.076,-62.356,-176.913,6.571,148.294
C00718=1218.179,255.325,-62.383,-176.911,6.574,148.294
C00719=1218.175,255.574,-62.410,-176.908,6.575,148.293
C00720=1218.170,255.822,-62.437,-176.906,6.578,148.293
C00721=1218.165,256.071,-62.464,-176.903,6.580,148.293
C00722=1218.161,256.319,-62.491,-176.901,6.581,148.293
C00723=1218.157,256.568,-62.518,-176.898,6.584,148.293
C00724=1218.152,256.816,-62.545,-176.895,6.586,148.292
C00725=1218.147,257.065,-62.572,-176.893,6.588,148.292
C00726=1218.144,257.313,-62.598,-176.891,6.590,148.292
C00727=1218.139,257.561,-62.625,-176.888,6.592,148.292
C00728=1218.134,257.810,-62.652,-176.886,6.594,148.292
C00729=1218.130,258.058,-62.680,-176.883,6.596,148.291
C00730=1218.126,258.307,-62.706,-176.880,6.599,148.291
C00731=1218.122,258.556,-62.733,-176.878,6.601,148.291
C00732=1218.117,258.804,-62.761,-176.875,6.603,148.291
C00733=1218.112,259.053,-62.788,-176.873,6.605,148.290
C00734=1218.108,259.301,-62.815,-176.871,6.607,148.290
C00735=1218.103,259.550,-62.842,-176.868,6.609,148.290
C00736=1218.099,259.798,-62.868,-176.865,6.612,148.290
C00737=1218.095,260.046,-62.896,-176.863,6.614,148.290
C00738=1218.091,260.295,-62.923,-176.861,6.616,148.289
C00739=1218.086,260.543,-62.950,-176.858,6.618,148.289
C00740=1218.081,260.792,-62.977,-176.856,6.620,148.289
C00741=1218.077,261.040,-63.005,-176.853,6.623,148.289
C00742=1218.072,261.289,-63.032,-176.850,6.625,148.288
C00743=1218.068,261.538,-63.059,-176.848,6.627,148.288
C00744=1218.064,261.786,-63.086,-176.845,6.629,148.288
C00745=1218.060,262.034,-63.113,-176.843,6.631,148.288
C00746=1218.055,262.283,-63.140,-176.840,6.634,148.288
C00747=1218.050,262.531,-63.167,-176.838,6.636,148.288
C00748=1218.047,262.780,-63.196,-176.835,6.638,148.287
C00749=1218.041,263.053,-63.225,-176.833,6.640,148.287
C00750=1218.037,263.325,-63.255,-176.830,6.643,148.287
C00751=1218.031,263.598,-63.285,-176.827,6.645,148.287
C00752=1218.027,263.870,-63.315,-176.824,6.647,148.286
C00753=1218.022,264.119,-63.342,-176.822,6.650,148.286
C00754=1218.018,264.367,-63.370,-176.819,6.651,148.286
C00755=1218.014,264.616,-63.397,-176.817,6.654,148.286
C00756=1218.009,264.864,-63.424,-176.814,6.656,148.286
C00757=1218.005,265.112,-63.452,-176.812,6.658,148.285
C00758=1218.001,265.361,-63.479,-176.809,6.660,148.285
C00759=1217.996,265.610,-63.506,-176.806,6.663,148.285
C00760=1217.992,265.858,-63.534,-176.804,6.665,148.285
C00761=1217.987,266.106,-63.561,-176.801,6.667,148.285
C00762=1217.983,266.355,-63.589,-176.799,6.669,148.285
C00763=1217.979,266.603,-63.617,-176.797,6.671,148.284
C00764=1217.974,266.852,-63.644,-176.794,6.674,148.284
C00765=1217.970,267.100,-63.672,-176.791,6.676,148.284
C00766=1217.966,267.349,-63.699,-176.789,6.678,148.284
C00767=1217.960,267.597,-63.727,-176.787,6.680,148.284
C00768=1217.956,267.845,-63.754,-176.784,6.683,148.284
C00769=1217.952,268.094,-63.782,-176.781,6.685,148.283
C00770=1217.947,268.342,-63.809,-176.779,6.687,148.283
C00771=1217.943,268.590,-63.837,-176.777,6.689,148.283
C00772=1217.939,268.840,-63.865,-176.774,6.692,148.283
C00773=1217.935,269.087,-63.892,-176.771,6.694,148.283
C00774=1217.930,269.336,-63.919,-176.769,6.696,148.283
C00775=1217.926,269.585,-63.948,-176.767,6.698,148.282
C00776=1217.921,269.833,-63.975,-176.764,6.701,148.282
C00777=1217.916,270.081,-64.003,-176.761,6.703,148.282
C00778=1217.912,270.330,-64.030,-176.759,6.705,148.282
C00779=1217.908,270.578,-64.058,-176.757,6.707,148.282
C00780=1217.904,270.826,-64.086,-176.754,6.710,148.282
C00781=1217.900,271.075,-64.113,-176.751,6.712,148.281
C00782=1217.895,271.324,-64.142,-176.749,6.714,148.281
C00783=1217.890,271.571,-64.170,-176.747,6.716,148.281
C00784=1217.886,271.821,-64.197,-176.744,6.719,148.281
C00785=1217.882,272.068,-64.225,-176.742,6.721,148.281
C00786=1217.877,272.317,-64.253,-176.739,6.723,148.280
C00787=1217.873,272.566,-64.281,-176.737,6.726,148.280
C00788=1217.868,272.814,-64.308,-176.734,6.728,148.280
C00789=1217.865,273.062,-64.337,-176.732,6.730,148.280
C00790=1217.859,273.311,-64.364,-176.729,6.732,148.280
C00791=1217.855,273.559,-64.392,-176.727,6.735,148.280
C00792=1217.851,273.808,-64.420,-176.724,6.737,148.279
C00793=1217.847,274.055,-64.448,-176.722,6.739,148.279
C00794=1217.842,274.305,-64.476,-176.719,6.741,148.279
C00795=1217.838,274.553,-64.504,-176.716,6.744,148.279
C00796=1217.834,274.801,-64.532,-176.714,6.747,148.279
C00797=1217.829,275.049,-64.560,-176.712,6.748,148.279
C00798=1217.824,275.297,-64.588,-176.710,6.751,148.279
C00799=1217.820,275.547,-64.615,-176.706,6.753,148.278
C00800=1217.816,275.795,-64.643,-176.704,6.756,148.278
C00801=1217.811,276.043,-64.672,-176.702,6.757,148.278
C00802=1217.807,276.291,-64.700,-176.699,6.760,148.278
C00803=1217.803,276.540,-64.728,-176.697,6.763,148.278
C00804=1217.798,276.788,-64.756,-176.694,6.765,148.278
C00805=1217.795,277.037,-64.784,-176.692,6.767,148.278
C00806=1217.789,277.285,-64.813,-176.689,6.769,148.277
C00807=1217.785,277.534,-64.840,-176.687,6.772,148.277
C00808=1217.781,277.782,-64.868,-176.685,6.774,148.277
C00809=1217.776,278.030,-64.896,-176.682,6.777,148.277
C00810=1217.772,278.279,-64.924,-176.680,6.779,148.277
C00811=1217.767,278.527,-64.953,-176.677,6.781,148.277
C00812=1217.763,278.775,-64.981,-176.674,6.784,148.276
C00813=1217.759,279.023,-65.009,-176.672,6.786,148.276
C00814=1217.755,279.272,-65.037,-176.670,6.788,148.276
C00815=1217.751,279.521,-65.066,-176.667,6.791,148.276
C00816=1217.746,279.769,-65.094,-176.665,6.793,148.276
C00817=1217.742,280.018,-65.122,-176.662,6.795,148.276
C00818=1217.737,280.266,-65.150,-176.660,6.797,148.276
C00819=1217.733,280.514,-65.179,-176.657,6.800,148.275
C00820=1217.728,280.762,-65.208,-176.655,6.802,148.275
C00821=1217.725,281.010,-65.236,-176.653,6.804,148.275
C00822=1217.719,281.259,-65.264,-176.649,6.807,148.275
C00823=1217.716,281.507,-65.292,-176.647,6.809,148.275
C00824=1217.711,281.755,-65.321,-176.645,6.811,148.275
C00825=1217.707,282.004,-65.349,-176.642,6.814,148.275
C00826=1217.702,282.253,-65.378,-176.640,6.816,148.275
C00827=1217.698,282.501,-65.405,-176.638,6.818,148.275
C00828=1217.694,282.749,-65.435,-176.635,6.821,148.274
C00829=1217.690,282.997,-65.463,-176.632,6.823,148.274
C00830=1217.685,283.246,-65.491,-176.630,6.826,148.274
C00831=1217.681,283.494,-65.519,-176.627,6.828,148.274
C00832=1217.676,283.743,-65.548,-176.625,6.831,148.274
C00833=1217.672,283.991,-65.577,-176.623,6.833,148.274
C00834=1217.668,284.239,-65.605,-176.620,6.835,148.274
C00835=1217.663,284.488,-65.634,-176.618,6.838,148.273
C00836=1217.659,284.735,-65.662,-176.616,6.840,148.273
C00837=1217.655,284.984,-65.691,-176.612,6.843,148.273
C00838=1217.650,285.233,-65.720,-176.610,6.845,148.273
C00839=1217.646,285.480,-65.748,-176.608,6.847,148.273
C00840=1217.641,285.729,-65.776,-176.605,6.850,148.273
C00841=1217.637,285.977,-65.805,-176.603,6.852,148.273
C00842=1217.633,286.225,-65.834,-176.601,6.854,148.273
C00843=1217.628,286.474,-65.862,-176.598,6.857,148.273
C00844=1217.624,286.722,-65.891,-176.595,6.859,148.272
C00845=1217.620,286.971,-65.920,-176.593,6.862,148.272
C00846=1217.616,287.219,-65.949,-176.591,6.864,148.272
C00847=1217.610,287.467,-65.977,-176.588,6.866,148.272
C00848=1217.607,287.716,-66.006,-176.585,6.869,148.272
C00849=1217.603,287.964,-66.035,-176.583,6.871,148.272
C00850=1217.597,288.212,-66.063,-176.581,6.874,148.272
C00851=1217.594,288.460,-66.092,-176.578,6.876,148.272
C00852=1217.590,288.709,-66.121,-176.576,6.879,148.271
C00853=1217.585,288.983,-66.153,-176.573,6.882,148.271
C00854=1217.580,289.257,-66.185,-176.571,6.883,148.271
C00855=1217.575,289.531,-66.217,-176.568,6.887,148.271
C00856=1217.570,289.805,-66.248,-176.565,6.890,148.271
C00857=1217.566,290.053,-66.277,-176.563,6.891,148.271
C00858=1217.561,290.302,-66.306,-176.560,6.894,148.271
C00859=1217.557,290.550,-66.335,-176.558,6.897,148.271
C00860=1217.553,290.798,-66.363,-176.556,6.899,148.271
C00861=1217.549,291.047,-66.393,-176.553,6.902,148.270
C00862=1217.544,291.295,-66.421,-176.551,6.904,148.270
C00863=1217.540,291.544,-66.451,-176.548,6.906,148.270
C00864=1217.535,291.791,-66.480,-176.546,6.909,148.270
C00865=1217.531,292.040,-66.508,-176.543,6.911,148.270
C00866=1217.527,292.288,-66.538,-176.540,6.914,148.270
C00867=1217.523,292.537,-66.566,-176.538,6.916,148.270
C00868=1217.518,292.785,-66.595,-176.536,6.918,148.270
C00869=1217.514,293.033,-66.625,-176.534,6.921,148.270
C00870=1217.509,293.282,-66.654,-176.531,6.923,148.270
C00871=1217.505,293.530,-66.683,-176.528,6.926,148.270
C00872=1217.501,293.777,-66.712,-176.526,6.929,148.270
C00873=1217.497,294.026,-66.740,-176.524,6.931,148.269
C00874=1217.492,294.274,-66.770,-176.521,6.934,148.269
C00875=1217.488,294.523,-66.799,-176.519,6.936,148.269
C00876=1217.484,294.771,-66.829,-176.516,6.939,148.269
C00877=1217.479,295.019,-66.857,-176.514,6.941,148.269
C00878=1217.475,295.267,-66.886,-176.512,6.943,148.269
C00879=1217.471,295.516,-66.916,-176.509,6.946,148.269
C00880=1217.466,295.764,-66.945,-176.507,6.948,148.269
C00881=1217.462,296.013,-66.974,-176.504,6.950,148.269
C00882=1217.457,296.260,-67.003,-176.502,6.953,148.269
C00883=1217.453,296.509,-67.033,-176.500,6.956,148.269
C00884=1217.449,296.757,-67.062,-176.497,6.959,148.269
C00885=1217.445,297.005,-67.092,-176.495,6.961,148.269
C00886=1217.440,297.253,-67.121,-176.492,6.964,148.269
C00887=1217.437,297.502,-67.149,-176.490,6.966,148.268
C00888=1217.432,297.750,-67.178,-176.487,6.968,148.268
C00889=1217.427,297.998,-67.208,-176.485,6.971,148.268
C00890=1217.423,298.246,-67.238,-176.483,6.973,148.268
C00891=1217.419,298.495,-67.267,-176.480,6.976,148.268
C00892=1217.414,298.743,-67.297,-176.478,6.978,148.268
C00893=1217.410,298.991,-67.326,-176.476,6.981,148.268
C00894=1217.406,299.239,-67.356,-176.473,6.984,148.268
C00895=1217.402,299.488,-67.385,-176.471,6.986,148.268
C00896=1217.397,299.735,-67.414,-176.468,6.989,148.268
C00897=1217.393,299.984,-67.444,-176.466,6.991,148.268
C00898=1217.389,300.232,-67.473,-176.464,6.993,148.268
C00899=1217.385,300.480,-67.502,-176.461,6.996,148.268
C00900=1217.380,300.728,-67.532,-176.459,6.998,148.267
C00901=1217.376,300.977,-67.561,-176.456,7.001,148.267
C00902=1217.372,301.225,-67.591,-176.454,7.004,148.267
C00903=1217.368,301.473,-67.620,-176.451,7.007,148.267
C00904=1217.363,301.722,-67.650,-176.449,7.009,148.267
C00905=1217.359,301.970,-67.680,-176.447,7.011,148.267
C00906=1217.355,302.218,-67.709,-176.444,7.014,148.267
C00907=1217.350,302.467,-67.739,-176.442,7.016,148.267
C00908=1217.346,302.714,-67.768,-176.440,7.019,148.267
C00909=1217.342,302.962,-67.798,-176.438,7.022,148.267
C00910=1217.337,303.210,-67.828,-176.435,7.025,148.267
C00911=1217.333,303.459,-67.857,-176.433,7.027,148.267
C00912=1217.328,303.707,-67.887,-176.430,7.029,148.267
C00913=1217.324,303.955,-67.916,-176.428,7.032,148.267
C00914=1217.320,304.203,-67.946,-176.425,7.034,148.267
C00915=1217.315,304.451,-67.977,-176.423,7.037,148.267
C00916=1217.311,304.700,-68.006,-176.421,7.039,148.267
C00917=1217.307,304.948,-68.035,-176.418,7.042,148.267
C00918=1217.303,305.196,-68.065,-176.416,7.044,148.267
C00919=1217.298,305.445,-68.095,-176.414,7.047,148.267
C00920=1217.294,305.692,-68.125,-176.411,7.050,148.267
C00921=1217.290,305.941,-68.155,-176.409,7.052,148.266
C00922=1217.286,306.189,-68.184,-176.406,7.055,148.266
C00923=1217.281,306.437,-68.215,-176.404,7.057,148.266
C00924=1217.277,306.685,-68.244,-176.401,7.060,148.266
C00925=1217.273,306.933,-68.274,-176.399,7.062,148.266
C00926=1217.269,307.182,-68.303,-176.397,7.065,148.266
C00927=1217.264,307.430,-68.334,-176.395,7.068,148.266
C00928=1217.260,307.678,-68.363,-176.392,7.070,148.266
C00929=1217.256,307.926,-68.393,-176.390,7.073,148.266
C00930=1217.251,308.174,-68.424,-176.388,7.075,148.266
C00931=1217.247,308.422,-68.453,-176.385,7.078,148.266
C00932=1217.243,308.670,-68.483,-176.383,7.081,148.266
C00933=1217.238,308.919,-68.513,-176.381,7.084,148.266
C00934=1217.234,309.167,-68.543,-176.379,7.086,148.266
C00935=1217.229,309.415,-68.574,-176.376,7.089,148.266
C00936=1217.226,309.664,-68.603,-176.374,7.091,148.266
C00937=1217.222,309.911,-68.633,-176.372,7.093,148.266
C00938=1217.217,310.160,-68.664,-176.369,7.096,148.266
C00939=1217.213,310.408,-68.694,-176.367,7.099,148.266
C00940=1217.209,310.656,-68.723,-176.364,7.102,148.266
C00941=1217.204,310.904,-68.754,-176.362,7.104,148.266
C00942=1217.200,311.152,-68.783,-176.359,7.107,148.266
C00943=1217.195,311.400,-68.814,-176.358,7.109,148.266
C00944=1217.191,311.648,-68.844,-176.355,7.112,148.266
C00945=1217.187,311.896,-68.874,-176.353,7.115,148.266
C00946=1217.182,312.145,-68.904,-176.350,7.118,148.266
C00947=1217.179,312.393,-68.934,-176.348,7.120,148.266
C00948=1217.175,312.641,-68.965,-176.346,7.122,148.266
C00949=1217.170,312.889,-68.995,-176.343,7.125,148.266
C00950=1217.166,313.137,-69.025,-176.341,7.127,148.266
C00951=1217.162,313.385,-69.055,-176.339,7.131,148.266
C00952=1217.157,313.633,-69.086,-176.337,7.133,148.266
C00953=1217.153,313.881,-69.116,-176.334,7.136,148.266
C00954=1217.149,314.130,-69.146,-176.332,7.138,148.266
C00955=1217.145,314.378,-69.176,-176.330,7.141,148.266
C00956=1217.140,314.626,-69.207,-176.327,7.143,148.266
C00957=1217.135,314.902,-69.241,-176.325,7.147,148.266
C00958=1217.131,315.178,-69.274,-176.322,7.150,148.266
C00959=1217.126,315.454,-69.308,-176.320,7.153,148.266
C00960=1217.121,315.730,-69.342,-176.317,7.156,148.266
C00961=1217.117,315.978,-69.372,-176.315,7.158,148.266
C00962=1217.112,316.226,-69.402,-176.312,7.161,148.266
C00963=1217.109,316.474,-69.433,-176.310,7.163,148.266
C00964=1217.104,316.722,-69.463,-176.308,7.166,148.266
C00965=1217.100,316.971,-69.494,-176.306,7.169,148.266
C00966=1217.096,317.219,-69.524,-176.304,7.171,148.266
C00967=1217.091,317.467,-69.555,-176.301,7.174,148.266
C00968=1217.087,317.714,-69.585,-176.299,7.176,148.266
C00969=1217.083,317.962,-69.616,-176.297,7.180,148.266
C00970=1217.079,318.211,-69.647,-176.295,7.182,148.266
C00971=1217.075,318.459,-69.677,-176.292,7.185,148.266
C00972=1217.070,318.707,-69.708,-176.290,7.187,148.266
C00973=1217.065,318.955,-69.738,-176.288,7.191,148.267
C00974=1217.062,319.204,-69.768,-176.286,7.193,148.267
C00975=1217.057,319.452,-69.799,-176.283,7.196,148.267
C00976=1217.053,319.699,-69.830,-176.281,7.198,148.266
C00977=1217.049,319.947,-69.860,-176.279,7.201,148.267
C00978=1217.045,320.196,-69.891,-176.277,7.204,148.267
C00979=1217.040,320.444,-69.922,-176.274,7.207,148.267
C00980=1217.036,320.691,-69.952,-176.272,7.209,148.267
C00981=1217.032,320.939,-69.983,-176.270,7.211,148.267
C00982=1217.028,321.188,-70.014,-176.268,7.215,148.267
C00983=1217.023,321.436,-70.045,-176.265,7.217,148.267
C00984=1217.019,321.684,-70.075,-176.263,7.220,148.267
C00985=1217.015,321.932,-70.106,-176.261,7.222,148.267
C00986=1217.011,322.180,-70.137,-176.259,7.225,148.267
C00987=1217.006,322.428,-70.167,-176.257,7.228,148.267
C00988=1217.003,322.677,-70.198,-176.254,7.231,148.267
C00989=1216.998,322.924,-70.229,-176.252,7.233,148.267
C00990=1216.994,323.172,-70.260,-176.250,7.236,148.267
C00991=1216.990,323.421,-70.291,-176.248,7.239,148.267
C00992=1216.986,323.669,-70.321,-176.245,7.242,148.267
C00993=1216.981,323.916,-70.352,-176.243,7.244,148.267
C00994=1216.977,324.165,-70.383,-176.241,7.247,148.267
C00995=1216.973,324.413,-70.414,-176.239,7.250,148.267
C00996=1216.968,324.661,-70.445,-176.237,7.253,148.268
C00997=1216.965,324.909,-70.476,-176.234,7.255,148.267
C00998=1216.960,325.157,-70.506,-176.232,7.258,148.268
C00999=1216.956,325.404,-70.538,-176.230,7.261,148.268
C01000=1216.952,325.653,-70.569,-176.227,7.264,148.268
C01001=1216.947,325.901,-70.600,-176.226,7.266,148.268
C01002=1216.943,326.149,-70.630,-176.224,7.268,148.268
C01003=1216.939,326.398,-70.662,-176.221,7.272,148.268
C01004=1216.935,326.645,-70.692,-176.219,7.274,148.268
C01005=1216.931,326.893,-70.724,-176.217,7.277,148.268
C01006=1216.926,327.141,-70.754,-176.215,7.280,148.268
C01007=1216.922,327.389,-70.785,-176.212,7.283,148.268
C01008=1216.918,327.637,-70.817,-176.211,7.285,148.268
C01009=1216.914,327.885,-70.848,-176.208,7.288,148.268
C01010=1216.910,328.134,-70.879,-176.206,7.291,148.268
C01011=1216.905,328.381,-70.910,-176.204,7.294,148.269
C01012=1216.901,328.629,-70.941,-176.202,7.296,148.269
C01013=1216.897,328.878,-70.972,-176.199,7.299,148.269
C01014=1216.892,329.125,-71.004,-176.198,7.302,148.269
C01015=1216.888,329.374,-71.035,-176.195,7.305,148.269
C01016=1216.884,329.621,-71.066,-176.194,7.307,148.269
C01017=1216.879,329.869,-71.097,-176.191,7.310,148.269
C01018=1216.875,330.118,-71.128,-176.189,7.313,148.269
C01019=1216.871,330.365,-71.160,-176.187,7.316,148.269
C01020=1216.867,330.614,-71.191,-176.185,7.319,148.269
C01021=1216.863,330.861,-71.222,-176.183,7.321,148.269
C01022=1216.859,331.110,-71.253,-176.181,7.324,148.270
C01023=1216.854,331.357,-71.285,-176.178,7.326,148.270
C01024=1216.850,331.606,-71.316,-176.176,7.330,148.270
C01025=1216.846,331.853,-71.347,-176.174,7.332,148.270
C01026=1216.842,332.102,-71.379,-176.172,7.335,148.270
C01027=1216.838,332.349,-71.410,-176.170,7.337,148.270
C01028=1216.834,332.598,-71.441,-176.168,7.341,148.270
C01029=1216.829,332.845,-71.473,-176.166,7.343,148.270
C01030=1216.825,333.094,-71.504,-176.163,7.346,148.270
C01031=1216.821,333.341,-71.535,-176.162,7.349,148.270
C01032=1216.817,333.590,-71.566,-176.159,7.352,148.270
C01033=1216.813,333.837,-71.598,-176.157,7.354,148.271
C01034=1216.809,334.086,-71.629,-176.155,7.358,148.271
C01035=1216.804,334.333,-71.661,-176.153,7.360,148.271
C01036=1216.800,334.581,-71.693,-176.151,7.363,148.271
C01037=1216.795,334.829,-71.724,-176.149,7.366,148.271
C01038=1216.792,335.077,-71.756,-176.147,7.368,148.271
C01039=1216.787,335.325,-71.787,-176.145,7.372,148.271
C01040=1216.783,335.573,-71.818,-176.143,7.374,148.271
C01041=1216.779,335.821,-71.850,-176.141,7.377,148.272
C01042=1216.775,336.069,-71.882,-176.139,7.380,148.272
C01043=1216.770,336.317,-71.913,-176.136,7.383,148.272
C01044=1216.766,336.565,-71.945,-176.135,7.385,148.272
C01045=1216.762,336.812,-71.976,-176.133,7.389,148.272
C01046=1216.758,337.061,-72.007,-176.130,7.391,148.272
C01047=1216.754,337.309,-72.040,-176.128,7.394,148.272
C01048=1216.749,337.557,-72.071,-176.127,7.397,148.273
C01049=1216.746,337.805,-72.103,-176.124,7.400,148.273
C01050=1216.741,338.053,-72.134,-176.122,7.402,148.273
C01051=1216.737,338.301,-72.166,-176.121,7.405,148.273
C01052=1216.732,338.548,-72.198,-176.118,7.408,148.273
C01053=1216.728,338.796,-72.230,-176.116,7.410,148.273
C01054=1216.725,339.044,-72.261,-176.114,7.414,148.273
C01055=1216.720,339.292,-72.292,-176.113,7.416,148.274
C01056=1216.716,339.541,-72.325,-176.110,7.419,148.274
C01057=1216.711,339.788,-72.356,-176.108,7.422,148.274
C01058=1216.708,340.036,-72.388,-176.106,7.425,148.274
C01059=1216.704,340.284,-72.420,-176.104,7.428,148.274
C01060=1216.699,340.532,-72.452,-176.102,7.431,148.274
C01061=1216.694,340.810,-72.487,-176.100,7.433,148.274
C01062=1216.689,341.088,-72.523,-176.098,7.437,148.275
C01063=1216.686,341.366,-72.559,-176.096,7.440,148.275
C01064=1216.680,341.644,-72.595,-176.093,7.443,148.275
C01065=1216.676,341.892,-72.626,-176.091,7.447,148.275
C01066=1216.672,342.140,-72.658,-176.089,7.449,148.275
C01067=1216.668,342.388,-72.690,-176.088,7.451,148.275
C01068=1216.663,342.636,-72.722,-176.085,7.455,148.276
C01069=1216.660,342.884,-72.754,-176.084,7.457,148.276
C01070=1216.655,343.132,-72.786,-176.082,7.461,148.276
C01071=1216.651,343.379,-72.817,-176.080,7.463,148.276
C01072=1216.647,343.628,-72.850,-176.077,7.466,148.276
C01073=1216.643,343.876,-72.882,-176.076,7.469,148.276
C01074=1216.639,344.123,-72.913,-176.074,7.471,148.277
C01075=1216.634,344.371,-72.946,-176.072,7.475,148.277
C01076=1216.631,344.619,-72.978,-176.070,7.477,148.277
C01077=1216.626,344.866,-73.010,-176.068,7.480,148.277
C01078=1216.622,345.115,-73.042,-176.066,7.483,148.277
C01079=1216.617,345.363,-73.075,-176.064,7.486,148.278
C01080=1216.613,345.610,-73.106,-176.062,7.489,148.278
C01081=1216.609,345.858,-73.138,-176.060,7.492,148.278
C01082=1216.605,346.107,-73.170,-176.059,7.495,148.278
C01083=1216.601,346.354,-73.202,-176.057,7.497,148.278
C01084=1216.597,346.602,-73.235,-176.054,7.500,148.278
C01085=1216.593,346.850,-73.267,-176.053,7.503,148.279
C01086=1216.588,347.098,-73.299,-176.050,7.506,148.279
C01087=1216.584,347.345,-73.331,-176.049,7.509,148.279
C01088=1216.580,347.594,-73.363,-176.047,7.512,148.279
C01089=1216.576,347.842,-73.395,-176.045,7.514,148.279
C01090=1216.572,348.090,-73.428,-176.043,7.517,148.280
C01091=1216.568,348.337,-73.460,-176.041,7.520,148.280
C01092=1216.563,348.585,-73.492,-176.039,7.523,148.280
C01093=1216.559,348.833,-73.524,-176.037,7.526,148.280
C01094=1216.555,349.081,-73.557,-176.036,7.529,148.280
C01095=1216.550,349.329,-73.589,-176.034,7.532,148.281
C01096=1216.546,349.577,-73.621,-176.032,7.535,148.281
C01097=1216.542,349.824,-73.654,-176.031,7.537,148.281
C01098=1216.539,350.072,-73.686,-176.028,7.541,148.281
C01099=1216.534,350.320,-73.718,-176.027,7.543,148.282
C01100=1216.530,350.567,-73.751,-176.025,7.546,148.282
C01101=1216.526,350.816,-73.783,-176.023,7.549,148.282
C01102=1216.521,351.064,-73.816,-176.021,7.552,148.282
C01103=1216.518,351.312,-73.848,-176.019,7.555,148.282
C01104=1216.513,351.559,-73.880,-176.017,7.558,148.283
C01105=1216.509,351.807,-73.912,-176.016,7.560,148.283
C01106=1216.505,352.055,-73.945,-176.014,7.563,148.283
C01107=1216.501,352.303,-73.978,-176.012,7.566,148.283
C01108=1216.497,352.551,-74.010,-176.010,7.570,148.284
C01109=1216.493,352.799,-74.043,-176.009,7.572,148.284
C01110=1216.488,353.047,-74.075,-176.007,7.575,148.284
C01111=1216.484,353.294,-74.107,-176.005,7.578,148.284
C01112=1216.480,353.543,-74.140,-176.003,7.581,148.284
C01113=1216.476,353.790,-74.173,-176.001,7.584,148.285
C01114=1216.472,354.038,-74.205,-176.000,7.587,148.285
C01115=1216.468,354.286,-74.238,-175.998,7.589,148.285
C01116=1216.463,354.534,-74.270,-175.996,7.593,148.285
C01117=1216.459,354.781,-74.303,-175.994,7.595,148.286
C01118=1216.455,355.029,-74.335,-175.992,7.599,148.286
C01119=1216.451,355.277,-74.368,-175.991,7.601,148.286
C01120=1216.447,355.525,-74.400,-175.989,7.604,148.286
C01121=1216.443,355.773,-74.433,-175.987,7.607,148.287
C01122=1216.439,356.021,-74.466,-175.986,7.610,148.287
C01123=1216.434,356.268,-74.498,-175.984,7.613,148.287
C01124=1216.430,356.516,-74.531,-175.982,7.616,148.287
C01125=1216.426,356.764,-74.563,-175.981,7.619,148.288
C01126=1216.422,357.012,-74.596,-175.979,7.621,148.288
C01127=1216.418,357.260,-74.630,-175.977,7.625,148.288
C01128=1216.414,357.508,-74.661,-175.975,7.627,148.288
C01129=1216.410,357.755,-74.695,-175.974,7.631,148.289
C01130=1216.406,358.003,-74.728,-175.972,7.633,148.289
C01131=1216.401,358.251,-74.760,-175.970,7.636,148.289
C01132=1216.397,358.499,-74.793,-175.969,7.639,148.290
C01133=1216.394,358.747,-74.826,-175.967,7.642,148.290
C01134=1216.389,358.994,-74.858,-175.965,7.644,148.290
C01135=1216.385,359.242,-74.891,-175.964,7.648,148.290
C01136=1216.380,359.490,-74.924,-175.962,7.651,148.291
C01137=1216.376,359.738,-74.957,-175.961,7.653,148.291
C01138=1216.373,359.985,-74.989,-175.959,7.657,148.291
C01139=1216.368,360.233,-75.023,-175.957,7.659,148.291
C01140=1216.364,360.481,-75.056,-175.956,7.662,148.292
C01141=1216.360,360.729,-75.088,-175.953,7.666,148.292
C01142=1216.356,360.977,-75.121,-175.952,7.668,148.292
C01143=1216.352,361.225,-75.154,-175.951,7.671,148.293
C01144=1216.347,361.472,-75.188,-175.949,7.674,148.293
C01145=1216.344,361.720,-75.220,-175.947,7.677,148.293
C01146=1216.340,361.968,-75.253,-175.946,7.680,148.294
C01147=1216.335,362.216,-75.286,-175.944,7.682,148.294
C01148=1216.331,362.464,-75.319,-175.943,7.686,148.294
C01149=1216.327,362.711,-75.352,-175.941,7.689,148.294
C01150=1216.323,362.959,-75.385,-175.940,7.691,148.295
C01151=1216.319,363.207,-75.418,-175.938,7.695,148.295
C01152=1216.315,363.455,-75.452,-175.936,7.698,148.296
C01153=1216.310,363.703,-75.484,-175.935,7.700,148.296
C01154=1216.306,363.951,-75.517,-175.934,7.703,148.296
C01155=1216.302,364.198,-75.550,-175.931,7.706,148.296
C01156=1216.299,364.446,-75.583,-175.930,7.709,148.297
C01157=1216.294,364.694,-75.616,-175.929,7.712,148.297
C01158=1216.290,364.941,-75.649,-175.927,7.714,148.297
C01159=1216.286,365.189,-75.682,-175.926,7.718,148.298
C01160=1216.282,365.437,-75.715,-175.924,7.721,148.298
C01161=1216.278,365.684,-75.749,-175.923,7.723,148.298
C01162=1216.274,365.932,-75.782,-175.922,7.726,148.299
C01163=1216.270,366.180,-75.815,-175.919,7.730,148.299
C01164=1216.266,366.428,-75.848,-175.918,7.732,148.299
C01165=1216.261,366.707,-75.886,-175.917,7.735,148.300
C01166=1216.256,366.988,-75.923,-175.915,7.739,148.300
C01167=1216.251,367.268,-75.961,-175.913,7.742,148.300
C01168=1216.247,367.548,-75.998,-175.912,7.745,148.301
C01169=1216.243,367.795,-76.032,-175.910,7.749,148.301
C01170=1216.238,368.043,-76.065,-175.909,7.751,148.301
C01171=1216.235,368.292,-76.098,-175.907,7.754,148.302
C01172=1216.231,368.539,-76.131,-175.906,7.757,148.302
C01173=1216.227,368.787,-76.165,-175.905,7.760,148.303
C01174=1216.222,369.035,-76.198,-175.903,7.762,148.303
C01175=1216.218,369.282,-76.231,-175.902,7.766,148.303
C01176=1216.214,369.530,-76.264,-175.900,7.769,148.304
C01177=1216.210,369.777,-76.298,-175.899,7.771,148.304
C01178=1216.205,370.025,-76.332,-175.898,7.774,148.304
C01179=1216.201,370.273,-76.365,-175.896,7.777,148.305
C01180=1216.197,370.521,-76.398,-175.895,7.780,148.305
C01181=1216.193,370.768,-76.431,-175.894,7.782,148.305
C01182=1216.189,371.016,-76.464,-175.892,7.786,148.306
C01183=1216.186,371.264,-76.499,-175.891,7.789,148.306
C01184=1216.182,371.512,-76.532,-175.890,7.791,148.306
C01185=1216.177,371.759,-76.565,-175.888,7.794,148.307
C01186=1216.173,372.008,-76.599,-175.887,7.797,148.307
C01187=1216.168,372.255,-76.632,-175.886,7.800,148.308
C01188=1216.165,372.502,-76.666,-175.885,7.803,148.308
C01189=1216.160,372.750,-76.699,-175.884,7.805,148.308
C01190=1216.156,372.998,-76.732,-175.882,7.808,148.309
C01191=1216.153,373.246,-76.765,-175.881,7.811,148.309
C01192=1216.149,373.493,-76.799,-175.879,7.815,148.310
C01193=1216.144,373.741,-76.833,-175.878,7.817,148.310
C01194=1216.140,373.989,-76.866,-175.877,7.820,148.310
C01195=1216.136,374.237,-76.899,-175.875,7.823,148.311
C01196=1216.132,374.484,-76.933,-175.874,7.826,148.311
C01197=1216.128,374.732,-76.966,-175.873,7.829,148.311
C01198=1216.124,374.980,-77.001,-175.872,7.831,148.312
C01199=1216.120,375.228,-77.034,-175.871,7.834,148.312
C01200=1216.116,375.475,-77.068,-175.869,7.837,148.313
C01201=1216.111,375.723,-77.101,-175.868,7.840,148.313
C01202=1216.108,375.970,-77.135,-175.867,7.843,148.313
C01203=1216.103,376.218,-77.168,-175.866,7.845,148.314
C01204=1216.099,376.466,-77.203,-175.865,7.848,148.314
C01205=1216.095,376.714,-77.236,-175.864,7.851,148.315
C01206=1216.091,376.961,-77.269,-175.862,7.854,148.315
C01207=1216.087,377.209,-77.303,-175.861,7.857,148.315
C01208=1216.082,377.457,-77.337,-175.860,7.860,148.316
C01209=1216.079,377.704,-77.371,-175.859,7.863,148.316
C01210=1216.074,377.952,-77.404,-175.858,7.865,148.317
C01211=1216.070,378.200,-77.438,-175.857,7.868,148.317
C01212=1216.066,378.447,-77.472,-175.856,7.871,148.318
C01213=1216.062,378.695,-77.505,-175.854,7.874,148.318
C01214=1216.058,378.943,-77.540,-175.854,7.876,148.318
C01215=1216.054,379.191,-77.573,-175.853,7.879,148.319
C01216=1216.050,379.438,-77.607,-175.851,7.881,148.319
C01217=1216.045,379.686,-77.640,-175.850,7.884,148.319
C01218=1216.042,379.933,-77.674,-175.850,7.887,148.320
C01219=1216.038,380.182,-77.708,-175.848,7.890,148.320
C01220=1216.034,380.429,-77.742,-175.847,7.893,148.321
C01221=1216.029,380.677,-77.775,-175.846,7.896,148.321
C01222=1216.026,380.924,-77.809,-175.845,7.899,148.322
C01223=1216.021,381.173,-77.843,-175.844,7.901,148.322
C01224=1216.017,381.420,-77.877,-175.843,7.904,148.323
C01225=1216.013,381.667,-77.910,-175.842,7.907,148.323
C01226=1216.009,381.915,-77.945,-175.841,7.909,148.323
C01227=1216.005,382.163,-77.979,-175.840,7.912,148.324
C01228=1216.001,382.410,-78.012,-175.839,7.915,148.324
C01229=1215.997,382.658,-78.047,-175.838,7.918,148.325
C01230=1215.993,382.905,-78.080,-175.837,7.920,148.325
C01231=1215.989,383.154,-78.115,-175.836,7.923,148.325
C01232=1215.985,383.401,-78.149,-175.835,7.926,148.326
C01233=1215.981,383.648,-78.182,-175.834,7.929,148.326
C01234=1215.976,383.896,-78.216,-175.833,7.932,148.327
C01235=1215.973,384.144,-78.250,-175.832,7.934,148.327
C01236=1215.968,384.392,-78.284,-175.832,7.937,148.328
C01237=1215.964,384.639,-78.318,-175.830,7.940,148.328
C01238=1215.960,384.887,-78.351,-175.829,7.942,148.329
C01239=1215.956,385.135,-78.386,-175.828,7.945,148.329
C01240=1215.952,385.382,-78.420,-175.828,7.947,148.330
C01241=1215.947,385.630,-78.454,-175.827,7.950,148.330
C01242=1215.944,385.878,-78.488,-175.825,7.953,148.330
C01243=1215.940,386.125,-78.522,-175.825,7.956,148.331
C01244=1215.935,386.373,-78.555,-175.824,7.958,148.331
C01245=1215.932,386.620,-78.589,-175.823,7.961,148.332
C01246=1215.928,386.868,-78.624,-175.822,7.964,148.332
C01247=1215.924,387.115,-78.658,-175.821,7.966,148.333
C01248=1215.919,387.363,-78.692,-175.820,7.969,148.333
C01249=1215.916,387.611,-78.726,-175.819,7.972,148.334
C01250=1215.911,387.858,-78.760,-175.818,7.975,148.334
C01251=1215.907,388.105,-78.794,-175.818,7.977,148.334
C01252=1215.903,388.354,-78.828,-175.817,7.980,148.335
C01253=1215.899,388.601,-78.862,-175.816,7.983,148.335
C01254=1215.895,388.849,-78.897,-175.816,7.985,148.336
C01255=1215.891,389.097,-78.931,-175.814,7.988,148.336
C01256=1215.887,389.344,-78.966,-175.813,7.991,148.337
C01257=1215.883,389.592,-78.999,-175.813,7.993,148.337
C01258=1215.879,389.840,-79.034,-175.812,7.996,148.338
C01259=1215.875,390.087,-79.067,-175.811,7.998,148.338
C01260=1215.870,390.334,-79.102,-175.810,8.001,148.338
C01261=1215.867,390.582,-79.136,-175.809,8.004,148.339
C01262=1215.863,390.830,-79.171,-175.809,8.006,148.339
C01263=1215.858,391.077,-79.204,-175.808,8.009,148.340
C01264=1215.854,391.325,-79.239,-175.808,8.011,148.340
C01265=1215.850,391.573,-79.273,-175.806,8.014,148.341
C01266=1215.846,391.820,-79.307,-175.805,8.017,148.341
C01267=1215.842,392.068,-79.342,-175.805,8.019,148.342
C01268=1215.838,392.315,-79.376,-175.804,8.022,148.342
C01269=1215.833,392.597,-79.414,-175.803,8.025,148.343
C01270=1215.829,392.880,-79.454,-175.802,8.028,148.343
C01271=1215.824,393.162,-79.492,-175.802,8.030,148.344
C01272=1215.819,393.443,-79.532,-175.801,8.033,148.344
C01273=1215.816,393.691,-79.566,-175.800,8.036,148.345
C01274=1215.812,393.939,-79.600,-175.800,8.038,148.345
C01275=1215.807,394.186,-79.635,-175.798,8.041,148.346
C01276=1215.804,394.434,-79.669,-175.798,8.043,148.346
C01277=1215.799,394.681,-79.704,-175.797,8.046,148.347
C01278=1215.796,394.929,-79.738,-175.797,8.048,148.347
C01279=1215.791,395.177,-79.772,-175.796,8.051,148.347
C01280=1215.787,395.425,-79.806,-175.795,8.053,148.348
C01281=1215.783,395.672,-79.840,-175.794,8.056,148.348
C01282=1215.779,395.920,-79.875,-175.794,8.058,148.349
C01283=1215.775,396.168,-79.910,-175.793,8.061,148.349
C01284=1215.771,396.415,-79.943,-175.793,8.064,148.350
C01285=1215.766,396.662,-79.978,-175.791,8.066,148.350
C01286=1215.763,396.910,-80.012,-175.791,8.069,148.351
C01287=1215.759,397.158,-80.047,-175.791,8.071,148.351
C01288=1215.755,397.406,-80.081,-175.790,8.074,148.352
C01289=1215.751,397.653,-80.115,-175.789,8.076,148.352
C01290=1215.747,397.900,-80.151,-175.788,8.079,148.353
C01291=1215.743,398.148,-80.185,-175.788,8.081,148.353
C01292=1215.739,398.395,-80.219,-175.788,8.083,148.354
C01293=1215.735,398.643,-80.254,-175.786,8.086,148.354
C01294=1215.730,398.890,-80.289,-175.786,8.088,148.354
C01295=1215.727,399.138,-80.323,-175.785,8.091,148.355
C01296=1215.722,399.386,-80.357,-175.785,8.093,148.355
C01297=1215.718,399.633,-80.392,-175.784,8.095,148.356
C01298=1215.715,399.881,-80.426,-175.783,8.098,148.356
C01299=1215.710,400.128,-80.460,-175.783,8.101,148.357
C01300=1215.706,400.376,-80.495,-175.783,8.103,148.357
C01301=1215.701,400.624,-80.530,-175.782,8.106,148.358
C01302=1215.698,400.872,-80.564,-175.781,8.108,148.358
C01303=1215.694,401.118,-80.599,-175.781,8.110,148.359
C01304=1215.690,401.367,-80.634,-175.780,8.113,148.359
C01305=1215.686,401.614,-80.668,-175.780,8.115,148.360
C01306=1215.682,401.862,-80.703,-175.779,8.117,148.360
C01307=1215.678,402.109,-80.737,-175.778,8.120,148.361
C01308=1215.673,402.357,-80.772,-175.778,8.122,148.361
C01309=1215.670,402.604,-80.806,-175.777,8.124,148.361
C01310=1215.666,402.851,-80.841,-175.776,8.127,148.362
C01311=1215.662,403.099,-80.876,-175.776,8.129,148.362
C01312=1215.657,403.347,-80.910,-175.776,8.132,148.363
C01313=1215.654,403.595,-80.945,-175.775,8.134,148.363
C01314=1215.649,403.842,-80.979,-175.774,8.137,148.364
C01315=1215.646,404.090,-81.015,-175.774,8.139,148.364
C01316=1215.641,404.337,-81.049,-175.773,8.141,148.365
C01317=1215.638,404.585,-81.083,-175.773,8.143,148.365
C01318=1215.633,404.832,-81.118,-175.772,8.146,148.366
C01319=1215.629,405.080,-81.153,-175.771,8.148,148.366
C01320=1215.625,405.327,-81.188,-175.771,8.150,148.367
C01321=1215.622,405.575,-81.222,-175.771,8.152,148.367
C01322=1215.617,405.822,-81.256,-175.770,8.155,148.367
C01323=1215.613,406.070,-81.291,-175.770,8.158,148.368
C01324=1215.609,406.317,-81.326,-175.769,8.160,148.368
C01325=1215.605,406.565,-81.361,-175.769,8.162,148.369
C01326=1215.601,406.812,-81.395,-175.768,8.164,148.369
C01327=1215.597,407.061,-81.430,-175.767,8.167,148.370
C01328=1215.593,407.307,-81.465,-175.767,8.169,148.370
C01329=1215.589,407.556,-81.500,-175.767,8.171,148.371
C01330=1215.584,407.803,-81.534,-175.766,8.173,148.371
C01331=1215.581,408.051,-81.569,-175.766,8.175,148.372
C01332=1215.577,408.298,-81.604,-175.765,8.178,148.372
C01333=1215.573,408.546,-81.639,-175.764,8.181,148.372
C01334=1215.568,408.793,-81.673,-175.764,8.183,148.373
C01335=1215.565,409.041,-81.709,-175.763,8.185,148.373
C01336=1215.561,409.288,-81.743,-175.763,8.187,148.374
C01337=1215.557,409.536,-81.777,-175.763,8.189,148.374
C01338=1215.553,409.783,-81.813,-175.762,8.191,148.375
C01339=1215.549,410.031,-81.847,-175.762,8.193,148.375
C01340=1215.544,410.278,-81.882,-175.762,8.196,148.376
C01341=1215.540,410.526,-81.917,-175.760,8.198,148.376
C01342=1215.536,410.773,-81.952,-175.760,8.201,148.377
C01343=1215.533,411.021,-81.986,-175.759,8.203,148.377
C01344=1215.529,411.268,-82.022,-175.759,8.205,148.377
C01345=1215.524,411.516,-82.056,-175.759,8.207,148.378
C01346=1215.520,411.764,-82.091,-175.758,8.209,148.378
C01347=1215.516,412.011,-82.126,-175.758,8.211,148.379
C01348=1215.512,412.259,-82.161,-175.758,8.213,148.379
C01349=1215.508,412.506,-82.196,-175.757,8.216,148.380
C01350=1215.505,412.753,-82.230,-175.757,8.218,148.380
C01351=1215.500,413.001,-82.265,-175.756,8.221,148.381
C01352=1215.496,413.248,-82.300,-175.755,8.223,148.381
C01353=1215.492,413.496,-82.335,-175.755,8.225,148.382
C01354=1215.488,413.743,-82.370,-175.754,8.227,148.382
C01355=1215.484,413.991,-82.405,-175.754,8.229,148.382
C01356=1215.480,414.239,-82.440,-175.754,8.231,148.383
C01357=1215.476,414.486,-82.475,-175.753,8.233,148.383
C01358=1215.471,414.734,-82.510,-175.753,8.235,148.384
C01359=1215.468,414.981,-82.545,-175.753,8.238,148.384
C01360=1215.464,415.228,-82.579,-175.752,8.240,148.384
C01361=1215.460,415.462,-82.612,-175.752,8.242,148.385
C01362=1215.456,415.694,-82.645,-175.751,8.244,148.385
C01363=1215.453,415.927,-82.678,-175.751,8.246,148.386
C01364=1215.448,416.160,-82.711,-175.750,8.248,148.386
C01365=1215.445,416.393,-82.745,-175.750,8.249,148.386
C01366=1215.441,416.625,-82.777,-175.750,8.252,148.387
C01367=1215.440,416.858,-82.810,-175.749,8.254,148.387
C01368=1215.440,417.091,-82.842,-175.749,8.255,148.388
C01369=1215.018,417.091,-82.878,-175.752,8.266,148.391
C01370=1215.017,416.857,-82.845,-175.753,8.264,148.391
C01371=1215.019,416.623,-82.812,-175.753,8.262,148.391
C01372=1215.023,416.389,-82.779,-175.753,8.260,148.390
C01373=1215.026,416.154,-82.746,-175.754,8.259,148.390
C01374=1215.031,415.920,-82.713,-175.754,8.257,148.389
C01375=1215.034,415.686,-82.680,-175.754,8.255,148.389
C01376=1215.039,415.452,-82.646,-175.755,8.252,148.389
C01377=1215.042,415.219,-82.614,-175.755,8.250,148.388
C01378=1215.046,414.970,-82.579,-175.756,8.248,148.388
C01379=1215.050,414.722,-82.544,-175.756,8.246,148.387
C01380=1215.055,414.476,-82.509,-175.756,8.244,148.387
C01381=1215.058,414.227,-82.474,-175.757,8.242,148.386
C01382=1215.062,413.981,-82.439,-175.757,8.240,148.386
C01383=1215.066,413.733,-82.404,-175.758,8.238,148.386
C01384=1215.070,413.486,-82.369,-175.758,8.235,148.385
C01385=1215.074,413.238,-82.334,-175.759,8.233,148.385
C01386=1215.078,412.990,-82.299,-175.759,8.230,148.384
C01387=1215.082,412.743,-82.264,-175.760,8.228,148.384
C01388=1215.086,412.495,-82.230,-175.760,8.226,148.383
C01389=1215.091,412.248,-82.194,-175.761,8.224,148.383
C01390=1215.095,412.000,-82.160,-175.761,8.222,148.382
C01391=1215.099,411.752,-82.125,-175.762,8.220,148.382
C01392=1215.102,411.505,-82.090,-175.762,8.217,148.382
C01393=1215.107,411.258,-82.056,-175.763,8.216,148.381
C01394=1215.110,411.010,-82.020,-175.763,8.213,148.381
C01395=1215.115,410.763,-81.986,-175.763,8.211,148.380
C01396=1215.119,410.515,-81.951,-175.764,8.209,148.380
C01397=1215.123,410.267,-81.915,-175.764,8.207,148.379
C01398=1215.127,410.020,-81.881,-175.765,8.204,148.379
C01399=1215.130,409.772,-81.847,-175.765,8.202,148.378
C01400=1215.135,409.525,-81.811,-175.766,8.200,148.378
C01401=1215.139,409.277,-81.777,-175.766,8.197,148.377
C01402=1215.143,409.030,-81.742,-175.767,8.195,148.377
C01403=1215.147,408.782,-81.707,-175.767,8.193,148.377
C01404=1215.151,408.535,-81.672,-175.767,8.191,148.376
C01405=1215.155,408.287,-81.638,-175.768,8.188,148.376
C01406=1215.159,408.040,-81.603,-175.769,8.186,148.375
C01407=1215.163,407.792,-81.568,-175.769,8.184,148.375
C01408=1215.167,407.545,-81.533,-175.769,8.182,148.374
C01409=1215.171,407.297,-81.498,-175.770,8.180,148.374
C01410=1215.175,407.050,-81.464,-175.770,8.177,148.373
C01411=1215.179,406.802,-81.429,-175.772,8.175,148.373
C01412=1215.183,406.555,-81.395,-175.772,8.172,148.372
C01413=1215.187,406.307,-81.359,-175.772,8.170,148.372
C01414=1215.192,406.060,-81.325,-175.773,8.168,148.372
C01415=1215.195,405.812,-81.290,-175.773,8.166,148.371
C01416=1215.200,405.564,-81.256,-175.774,8.163,148.371
C01417=1215.203,405.317,-81.220,-175.774,8.161,148.370
C01418=1215.208,405.069,-81.186,-175.775,8.159,148.370
C01419=1215.212,404.821,-81.151,-175.775,8.156,148.369
C01420=1215.216,404.574,-81.117,-175.776,8.154,148.369
C01421=1215.219,404.327,-81.082,-175.776,8.151,148.368
C01422=1215.224,404.079,-81.047,-175.777,8.149,148.368
C01423=1215.228,403.831,-81.012,-175.777,8.147,148.367
C01424=1215.232,403.584,-80.978,-175.778,8.144,148.367
C01425=1215.236,403.336,-80.944,-175.779,8.142,148.366
C01426=1215.240,403.089,-80.908,-175.779,8.140,148.366
C01427=1215.244,402.841,-80.874,-175.780,8.138,148.366
C01428=1215.248,402.594,-80.840,-175.780,8.135,148.365
C01429=1215.252,402.346,-80.805,-175.781,8.133,148.365
C01430=1215.256,402.098,-80.770,-175.781,8.130,148.364
C01431=1215.260,401.850,-80.736,-175.782,8.127,148.364
C01432=1215.264,401.603,-80.702,-175.783,8.125,148.363
C01433=1215.268,401.356,-80.667,-175.783,8.123,148.363
C01434=1215.272,401.108,-80.632,-175.783,8.121,148.362
C01435=1215.276,400.861,-80.598,-175.784,8.118,148.362
C01436=1215.280,400.613,-80.563,-175.785,8.116,148.361
C01437=1215.285,400.366,-80.529,-175.785,8.114,148.361
C01438=1215.289,400.117,-80.494,-175.786,8.111,148.360
C01439=1215.292,399.870,-80.460,-175.786,8.109,148.360
C01440=1215.296,399.622,-80.425,-175.787,8.107,148.360
C01441=1215.301,399.375,-80.390,-175.788,8.104,148.359
C01442=1215.304,399.128,-80.356,-175.788,8.101,148.358
C01443=1215.308,398.880,-80.321,-175.789,8.098,148.358
C01444=1215.313,398.633,-80.287,-175.789,8.096,148.357
C01445=1215.316,398.385,-80.252,-175.790,8.094,148.357
C01446=1215.321,398.138,-80.218,-175.791,8.091,148.357
C01447=1215.325,397.889,-80.183,-175.791,8.089,148.356
C01448=1215.329,397.642,-80.149,-175.792,8.086,148.356
C01449=1215.333,397.395,-80.115,-175.793,8.084,148.355
C01450=1215.337,397.147,-80.080,-175.793,8.082,148.355
C01451=1215.341,396.900,-80.046,-175.794,8.079,148.354
C01452=1215.345,396.652,-80.011,-175.794,8.077,148.354
C01453=1215.349,396.404,-79.977,-175.796,8.074,148.353
C01454=1215.353,396.156,-79.943,-175.796,8.072,148.353
C01455=1215.357,395.909,-79.908,-175.797,8.069,148.352
C01456=1215.362,395.662,-79.874,-175.797,8.067,148.352
C01457=1215.365,395.414,-79.839,-175.798,8.064,148.352
C01458=1215.370,395.166,-79.805,-175.799,8.061,148.351
C01459=1215.373,394.918,-79.771,-175.800,8.059,148.351
C01460=1215.377,394.671,-79.736,-175.800,8.056,148.350
C01461=1215.382,394.424,-79.702,-175.801,8.054,148.350
C01462=1215.385,394.176,-79.668,-175.801,8.051,148.349
C01463=1215.390,393.928,-79.633,-175.803,8.048,148.349
C01464=1215.394,393.681,-79.599,-175.803,8.046,148.348
C01465=1215.398,393.433,-79.564,-175.804,8.043,148.348
C01466=1215.403,393.151,-79.526,-175.804,8.041,148.347
C01467=1215.407,392.870,-79.487,-175.805,8.038,148.347
C01468=1215.412,392.587,-79.448,-175.806,8.035,148.346
C01469=1215.416,392.305,-79.408,-175.807,8.032,148.346
C01470=1215.420,392.058,-79.374,-175.808,8.029,148.345
C01471=1215.424,391.810,-79.340,-175.808,8.027,148.345
C01472=1215.428,391.563,-79.306,-175.809,8.024,148.344
C01473=1215.432,391.315,-79.271,-175.810,8.022,148.344
C01474=1215.437,391.066,-79.237,-175.811,8.019,148.343
C01475=1215.441,390.819,-79.203,-175.812,8.016,148.343
C01476=1215.445,390.571,-79.168,-175.812,8.014,148.342
C01477=1215.449,390.324,-79.134,-175.813,8.011,148.342
C01478=1215.453,390.077,-79.100,-175.814,8.009,148.342
C01479=1215.456,389.829,-79.066,-175.815,8.006,148.341
C01480=1215.461,389.581,-79.032,-175.815,8.003,148.341
C01481=1215.465,389.334,-78.998,-175.816,8.001,148.340
C01482=1215.469,389.086,-78.963,-175.817,7.998,148.340
C01483=1215.473,388.839,-78.929,-175.818,7.995,148.339
C01484=1215.477,388.591,-78.895,-175.819,7.993,148.339
C01485=1215.481,388.343,-78.861,-175.819,7.990,148.338
C01486=1215.486,388.095,-78.827,-175.821,7.987,148.338
C01487=1215.489,387.848,-78.793,-175.821,7.985,148.338
C01488=1215.493,387.600,-78.758,-175.822,7.982,148.337
C01489=1215.497,387.353,-78.724,-175.823,7.979,148.337
C01490=1215.502,387.105,-78.691,-175.824,7.977,148.336
C01491=1215.505,386.857,-78.656,-175.825,7.974,148.336
C01492=1215.510,386.610,-78.622,-175.826,7.971,148.335
C01493=1215.514,386.362,-78.589,-175.827,7.968,148.335
C01494=1215.518,386.114,-78.554,-175.827,7.966,148.334
C01495=1215.522,385.867,-78.520,-175.828,7.963,148.334
C01496=1215.526,385.620,-78.486,-175.830,7.961,148.333
C01497=1215.530,385.372,-78.452,-175.830,7.958,148.333
C01498=1215.534,385.124,-78.418,-175.831,7.956,148.333
C01499=1215.538,384.876,-78.384,-175.832,7.953,148.332
C01500=1215.542,384.629,-78.351,-175.833,7.950,148.332
C01501=1215.546,384.380,-78.316,-175.834,7.947,148.331
C01502=1215.550,384.133,-78.282,-175.835,7.945,148.331
C01503=1215.554,383.886,-78.249,-175.835,7.942,148.330
C01504=1215.559,383.638,-78.214,-175.837,7.939,148.330
C01505=1215.562,383.390,-78.180,-175.838,7.936,148.329
C01506=1215.567,383.142,-78.146,-175.839,7.933,148.329
C01507=1215.571,382.895,-78.112,-175.839,7.931,148.328
C01508=1215.575,382.648,-78.079,-175.840,7.928,148.328
C01509=1215.579,382.399,-78.044,-175.842,7.925,148.328
C01510=1215.583,382.152,-78.011,-175.843,7.923,148.327
C01511=1215.588,381.904,-77.977,-175.844,7.919,148.327
C01512=1215.591,381.657,-77.943,-175.845,7.917,148.326
C01513=1215.595,381.409,-77.909,-175.846,7.914,148.326
C01514=1215.600,381.161,-77.875,-175.847,7.912,148.326
C01515=1215.604,380.914,-77.842,-175.848,7.909,148.325
C01516=1215.608,380.666,-77.808,-175.849,7.906,148.325
C01517=1215.612,380.418,-77.774,-175.850,7.903,148.324
C01518=1215.616,380.171,-77.740,-175.851,7.900,148.324
C01519=1215.620,379.923,-77.707,-175.852,7.897,148.323
C01520=1215.624,379.675,-77.672,-175.853,7.895,148.323
C01521=1215.628,379.427,-77.639,-175.854,7.892,148.323
C01522=1215.632,379.180,-77.605,-175.855,7.889,148.322
C01523=1215.637,378.932,-77.571,-175.856,7.886,148.322
C01524=1215.640,378.685,-77.537,-175.857,7.884,148.321
C01525=1215.645,378.437,-77.504,-175.858,7.881,148.321
C01526=1215.649,378.189,-77.469,-175.859,7.878,148.321
C01527=1215.653,377.941,-77.436,-175.861,7.875,148.320
C01528=1215.657,377.694,-77.402,-175.862,7.873,148.320
C01529=1215.661,377.446,-77.369,-175.863,7.870,148.319
C01530=1215.665,377.199,-77.335,-175.864,7.867,148.319
C01531=1215.669,376.951,-77.301,-175.865,7.864,148.319
C01532=1215.673,376.703,-77.268,-175.867,7.861,148.318
C01533=1215.677,376.456,-77.234,-175.868,7.859,148.318
C01534=1215.682,376.208,-77.200,-175.868,7.855,148.317
C01535=1215.685,375.961,-77.167,-175.870,7.853,148.317
C01536=1215.690,375.713,-77.133,-175.871,7.850,148.316
C01537=1215.693,375.464,-77.100,-175.872,7.847,148.316
C01538=1215.698,375.217,-77.065,-175.873,7.844,148.316
C01539=1215.702,374.969,-77.032,-175.874,7.841,148.315
C01540=1215.706,374.721,-76.999,-175.876,7.839,148.315
C01541=1215.710,374.474,-76.965,-175.877,7.836,148.314
C01542=1215.714,374.227,-76.932,-175.878,7.833,148.314
C01543=1215.718,373.978,-76.898,-175.880,7.830,148.314
C01544=1215.722,373.731,-76.864,-175.881,7.828,148.313
C01545=1215.726,373.483,-76.831,-175.883,7.824,148.313
C01546=1215.730,373.235,-76.798,-175.884,7.821,148.313
C01547=1215.734,372.988,-76.765,-175.885,7.818,148.312
C01548=1215.739,372.740,-76.730,-175.886,7.816,148.312
C01549=1215.743,372.492,-76.697,-175.887,7.813,148.311
C01550=1215.747,372.244,-76.663,-175.889,7.810,148.311
C01551=1215.751,371.996,-76.630,-175.890,7.807,148.311
C01552=1215.755,371.749,-76.596,-175.891,7.804,148.310
C01553=1215.759,371.501,-76.563,-175.892,7.801,148.310
C01554=1215.763,371.254,-76.530,-175.894,7.799,148.310
C01555=1215.768,371.006,-76.496,-175.896,7.795,148.309
C01556=1215.772,370.758,-76.463,-175.897,7.792,148.309
C01557=1215.776,370.511,-76.429,-175.898,7.790,148.308
C01558=1215.780,370.263,-76.396,-175.899,7.787,148.308
C01559=1215.783,370.015,-76.363,-175.900,7.784,148.308
C01560=1215.788,369.767,-76.329,-175.902,7.781,148.307
C01561=1215.792,369.519,-76.296,-175.903,7.779,148.307
C01562=1215.796,369.272,-76.263,-175.905,7.775,148.307
C01563=1215.800,369.024,-76.229,-175.906,7.772,148.306
C01564=1215.804,368.777,-76.196,-175.908,7.770,148.306
C01565=1215.809,368.529,-76.162,-175.909,7.767,148.306
C01566=1215.813,368.281,-76.129,-175.910,7.764,148.305
C01567=1215.817,368.033,-76.096,-175.912,7.760,148.305
C01568=1215.821,367.785,-76.063,-175.913,7.758,148.305
C01569=1215.825,367.538,-76.030,-175.915,7.755,148.304
C01570=1215.829,367.257,-75.992,-175.916,7.751,148.304
C01571=1215.834,366.977,-75.955,-175.918,7.749,148.303
C01572=1215.839,366.698,-75.918,-175.920,7.745,148.303
C01573=1215.843,366.417,-75.880,-175.921,7.742,148.303
C01574=1215.847,366.170,-75.846,-175.923,7.739,148.302
C01575=1215.851,365.922,-75.813,-175.924,7.736,148.302
C01576=1215.855,365.674,-75.780,-175.925,7.733,148.302
C01577=1215.859,365.426,-75.747,-175.927,7.731,148.301
C01578=1215.863,365.179,-75.714,-175.929,7.727,148.301
C01579=1215.868,364.931,-75.681,-175.930,7.724,148.301
C01580=1215.872,364.683,-75.648,-175.931,7.722,148.300
C01581=1215.876,364.436,-75.614,-175.933,7.719,148.300
C01582=1215.880,364.188,-75.581,-175.935,7.715,148.300
C01583=1215.884,363.940,-75.548,-175.936,7.713,148.299
C01584=1215.889,363.692,-75.516,-175.937,7.710,148.299
C01585=1215.893,363.444,-75.482,-175.940,7.707,148.299
C01586=1215.897,363.196,-75.449,-175.941,7.704,148.298
C01587=1215.901,362.949,-75.416,-175.943,7.701,148.298
C01588=1215.905,362.701,-75.383,-175.944,7.699,148.298
C01589=1215.909,362.453,-75.350,-175.946,7.695,148.298
C01590=1215.913,362.205,-75.317,-175.947,7.692,148.297
C01591=1215.917,361.958,-75.284,-175.949,7.690,148.297
C01592=1215.921,361.710,-75.252,-175.950,7.686,148.297
C01593=1215.925,361.462,-75.219,-175.952,7.684,148.296
C01594=1215.930,361.214,-75.185,-175.953,7.681,148.296
C01595=1215.934,360.966,-75.152,-175.955,7.678,148.296
C01596=1215.938,360.719,-75.119,-175.957,7.675,148.295
C01597=1215.942,360.470,-75.087,-175.958,7.672,148.295
C01598=1215.946,360.223,-75.053,-175.960,7.669,148.295
C01599=1215.950,359.975,-75.021,-175.962,7.666,148.295
C01600=1215.954,359.727,-74.988,-175.963,7.664,148.294
C01601=1215.958,359.479,-74.955,-175.965,7.660,148.294
C01602=1215.963,359.232,-74.923,-175.967,7.657,148.294
C01603=1215.967,358.984,-74.889,-175.968,7.655,148.293
C01604=1215.971,358.737,-74.856,-175.970,7.651,148.293
C01605=1215.975,358.489,-74.824,-175.972,7.649,148.293
C01606=1215.979,358.241,-74.791,-175.973,7.646,148.293
C01607=1215.983,357.993,-74.758,-175.975,7.643,148.292
C01608=1215.988,357.745,-74.726,-175.977,7.640,148.292
C01609=1215.991,357.497,-74.693,-175.978,7.637,148.292
C01610=1215.995,357.250,-74.660,-175.980,7.634,148.292
C01611=1216.000,357.001,-74.627,-175.982,7.631,148.291
C01612=1216.004,356.753,-74.594,-175.983,7.628,148.291
C01613=1216.008,356.505,-74.562,-175.985,7.625,148.291
C01614=1216.012,356.258,-74.530,-175.987,7.623,148.291
C01615=1216.017,356.011,-74.497,-175.989,7.619,148.290
C01616=1216.021,355.762,-74.464,-175.990,7.616,148.290
C01617=1216.024,355.515,-74.432,-175.992,7.614,148.290
C01618=1216.029,355.267,-74.399,-175.994,7.611,148.290
C01619=1216.033,355.019,-74.366,-175.996,7.608,148.289
C01620=1216.037,354.770,-74.333,-175.997,7.605,148.289
C01621=1216.041,354.523,-74.301,-175.999,7.602,148.289
C01622=1216.046,354.275,-74.269,-176.001,7.599,148.289
C01623=1216.050,354.028,-74.236,-176.003,7.596,148.288
C01624=1216.054,353.780,-74.204,-176.004,7.593,148.288
C01625=1216.058,353.532,-74.171,-176.006,7.591,148.288
C01626=1216.062,353.284,-74.138,-176.008,7.587,148.288
C01627=1216.066,353.036,-74.106,-176.010,7.585,148.287
C01628=1216.071,352.789,-74.074,-176.012,7.581,148.287
C01629=1216.075,352.541,-74.040,-176.013,7.579,148.287
C01630=1216.079,352.293,-74.009,-176.015,7.576,148.287
C01631=1216.083,352.045,-73.975,-176.017,7.573,148.286
C01632=1216.087,351.797,-73.943,-176.018,7.570,148.286
C01633=1216.091,351.549,-73.911,-176.021,7.567,148.286
C01634=1216.096,351.302,-73.878,-176.022,7.564,148.286
C01635=1216.099,351.054,-73.847,-176.024,7.562,148.286
C01636=1216.104,350.805,-73.814,-176.026,7.558,148.285
C01637=1216.108,350.557,-73.781,-176.028,7.556,148.285
C01638=1216.112,350.309,-73.749,-176.030,7.553,148.285
C01639=1216.117,350.062,-73.717,-176.031,7.550,148.284
C01640=1216.120,349.814,-73.684,-176.033,7.547,148.284
C01641=1216.125,349.566,-73.652,-176.035,7.544,148.284
C01642=1216.129,349.318,-73.620,-176.037,7.541,148.284
C01643=1216.133,349.071,-73.587,-176.039,7.538,148.284
C01644=1216.137,348.823,-73.555,-176.040,7.536,148.283
C01645=1216.141,348.575,-73.523,-176.043,7.532,148.283
C01646=1216.146,348.326,-73.491,-176.044,7.530,148.283
C01647=1216.150,348.080,-73.458,-176.046,7.527,148.283
C01648=1216.154,347.831,-73.426,-176.048,7.524,148.283
C01649=1216.158,347.583,-73.394,-176.050,7.521,148.282
C01650=1216.162,347.335,-73.362,-176.052,7.518,148.282
C01651=1216.166,347.088,-73.330,-176.054,7.515,148.282
C01652=1216.171,346.840,-73.297,-176.056,7.512,148.282
C01653=1216.174,346.592,-73.265,-176.057,7.510,148.282
C01654=1216.179,346.343,-73.233,-176.059,7.507,148.282
C01655=1216.183,346.096,-73.201,-176.061,7.504,148.281
C01656=1216.187,345.848,-73.169,-176.063,7.501,148.281
C01657=1216.191,345.600,-73.136,-176.065,7.498,148.281
C01658=1216.196,345.353,-73.104,-176.067,7.496,148.281
C01659=1216.200,345.105,-73.072,-176.069,7.492,148.281
C01660=1216.204,344.856,-73.040,-176.071,7.490,148.280
C01661=1216.208,344.608,-73.008,-176.073,7.486,148.280
C01662=1216.212,344.361,-72.977,-176.075,7.484,148.280
C01663=1216.217,344.112,-72.944,-176.077,7.481,148.280
C01664=1216.220,343.864,-72.912,-176.079,7.478,148.280
C01665=1216.225,343.617,-72.880,-176.080,7.475,148.280
C01666=1216.229,343.369,-72.848,-176.083,7.472,148.279
C01667=1216.233,343.121,-72.817,-176.084,7.470,148.279
C01668=1216.238,342.873,-72.785,-176.087,7.466,148.279
C01669=1216.241,342.625,-72.753,-176.089,7.464,148.279
C01670=1216.246,342.377,-72.720,-176.091,7.461,148.279
C01671=1216.250,342.129,-72.689,-176.092,7.458,148.279
C01672=1216.254,341.881,-72.657,-176.094,7.456,148.278
C01673=1216.259,341.634,-72.625,-176.096,7.452,148.278
C01674=1216.263,341.355,-72.589,-176.099,7.449,148.278
C01675=1216.268,341.078,-72.553,-176.101,7.446,148.278
C01676=1216.272,340.799,-72.518,-176.103,7.442,148.278
C01677=1216.277,340.522,-72.482,-176.105,7.440,148.277
C01678=1216.282,340.274,-72.450,-176.108,7.437,148.277
C01679=1216.285,340.026,-72.418,-176.109,7.434,148.277
C01680=1216.289,339.778,-72.386,-176.111,7.431,148.277
C01681=1216.294,339.530,-72.355,-176.113,7.428,148.277
C01682=1216.298,339.282,-72.323,-176.115,7.425,148.277
C01683=1216.302,339.034,-72.291,-176.117,7.423,148.277
C01684=1216.306,338.786,-72.260,-176.120,7.420,148.276
C01685=1216.311,338.538,-72.227,-176.121,7.417,148.276
C01686=1216.315,338.291,-72.196,-176.124,7.414,148.276
C01687=1216.319,338.042,-72.165,-176.126,7.411,148.276
C01688=1216.323,337.794,-72.133,-176.127,7.409,148.276
C01689=1216.328,337.546,-72.101,-176.129,7.406,148.276
C01690=1216.331,337.298,-72.069,-176.131,7.403,148.276
C01691=1216.336,337.050,-72.038,-176.134,7.400,148.275
C01692=1216.340,336.802,-72.006,-176.135,7.398,148.275
C01693=1216.344,336.555,-71.975,-176.138,7.394,148.275
C01694=1216.348,336.307,-71.943,-176.140,7.392,148.275
C01695=1216.353,336.059,-71.912,-176.142,7.389,148.275
C01696=1216.357,335.811,-71.880,-176.144,7.386,148.275
C01697=1216.361,335.563,-71.848,-176.146,7.383,148.275
C01698=1216.365,335.315,-71.817,-176.148,7.381,148.275
C01699=1216.369,335.067,-71.785,-176.150,7.377,148.275
C01700=1216.374,334.819,-71.753,-176.152,7.375,148.274
C01701=1216.378,334.570,-71.722,-176.154,7.372,148.274
C01702=1216.382,334.323,-71.691,-176.156,7.369,148.274
C01703=1216.386,334.074,-71.660,-176.159,7.366,148.274
C01704=1216.391,333.827,-71.628,-176.161,7.364,148.274
C01705=1216.394,333.579,-71.596,-176.163,7.360,148.274
C01706=1216.399,333.331,-71.566,-176.165,7.358,148.274
C01707=1216.403,333.083,-71.534,-176.167,7.356,148.274
C01708=1216.407,332.835,-71.503,-176.169,7.352,148.273
C01709=1216.411,332.587,-71.471,-176.171,7.350,148.273
C01710=1216.416,332.339,-71.440,-176.173,7.347,148.273
C01711=1216.420,332.091,-71.408,-176.175,7.345,148.273
C01712=1216.425,331.843,-71.377,-176.177,7.341,148.273
C01713=1216.428,331.595,-71.345,-176.179,7.339,148.273
C01714=1216.433,331.347,-71.315,-176.182,7.336,148.273
C01715=1216.437,331.099,-71.283,-176.183,7.333,148.273
C01716=1216.441,330.851,-71.252,-176.186,7.330,148.273
C01717=1216.445,330.603,-71.220,-176.188,7.328,148.273
C01718=1216.450,330.355,-71.189,-176.190,7.325,148.273
C01719=1216.454,330.107,-71.158,-176.192,7.322,148.272
C01720=1216.458,329.859,-71.127,-176.195,7.319,148.272
C01721=1216.462,329.611,-71.096,-176.196,7.316,148.272
C01722=1216.466,329.363,-71.064,-176.199,7.313,148.272
C01723=1216.471,329.115,-71.033,-176.201,7.311,148.272
C01724=1216.474,328.867,-71.001,-176.203,7.308,148.272
C01725=1216.479,328.619,-70.971,-176.205,7.305,148.272
C01726=1216.484,328.371,-70.940,-176.208,7.302,148.272
C01727=1216.487,328.123,-70.908,-176.209,7.300,148.272
C01728=1216.492,327.875,-70.877,-176.212,7.297,148.272
C01729=1216.495,327.626,-70.847,-176.214,7.294,148.271
C01730=1216.500,327.379,-70.815,-176.216,7.292,148.271
C01731=1216.504,327.131,-70.785,-176.218,7.289,148.271
C01732=1216.508,326.883,-70.753,-176.220,7.286,148.271
C01733=1216.513,326.635,-70.723,-176.223,7.283,148.271
C01734=1216.517,326.387,-70.691,-176.224,7.281,148.271
C01735=1216.521,326.139,-70.660,-176.227,7.278,148.271
C01736=1216.526,325.891,-70.629,-176.229,7.275,148.271
C01737=1216.530,325.642,-70.598,-176.231,7.272,148.271
C01738=1216.533,325.395,-70.567,-176.233,7.270,148.271
C01739=1216.538,325.147,-70.537,-176.236,7.267,148.271
C01740=1216.542,324.898,-70.505,-176.238,7.264,148.271
C01741=1216.547,324.650,-70.475,-176.240,7.261,148.271
C01742=1216.551,324.402,-70.444,-176.242,7.259,148.271
C01743=1216.555,324.154,-70.413,-176.245,7.256,148.271
C01744=1216.559,323.907,-70.382,-176.246,7.253,148.270
C01745=1216.563,323.659,-70.351,-176.249,7.250,148.270
C01746=1216.567,323.410,-70.320,-176.251,7.248,148.271
C01747=1216.572,323.162,-70.289,-176.253,7.245,148.270
C01748=1216.577,322.914,-70.258,-176.255,7.242,148.270
C01749=1216.580,322.666,-70.228,-176.258,7.239,148.270
C01750=1216.585,322.418,-70.197,-176.260,7.237,148.270
C01751=1216.589,322.170,-70.166,-176.262,7.234,148.270
C01752=1216.593,321.921,-70.135,-176.264,7.232,148.270
C01753=1216.597,321.674,-70.105,-176.267,7.228,148.270
C01754=1216.602,321.426,-70.074,-176.269,7.226,148.270
C01755=1216.606,321.177,-70.043,-176.271,7.223,148.270
C01756=1216.610,320.929,-70.013,-176.273,7.221,148.270
C01757=1216.614,320.681,-69.982,-176.275,7.218,148.270
C01758=1216.619,320.433,-69.951,-176.278,7.215,148.270
C01759=1216.623,320.185,-69.920,-176.280,7.213,148.270
C01760=1216.627,319.937,-69.890,-176.282,7.210,148.270
C01761=1216.631,319.689,-69.859,-176.284,7.207,148.270
C01762=1216.635,319.440,-69.828,-176.287,7.204,148.270
C01763=1216.639,319.193,-69.798,-176.289,7.202,148.270
C01764=1216.644,318.945,-69.767,-176.291,7.199,148.270
C01765=1216.648,318.697,-69.737,-176.293,7.197,148.270
C01766=1216.652,318.449,-69.706,-176.296,7.194,148.270
C01767=1216.657,318.200,-69.676,-176.298,7.191,148.270
C01768=1216.661,317.952,-69.645,-176.300,7.188,148.270
C01769=1216.665,317.704,-69.615,-176.302,7.186,148.270
C01770=1216.670,317.456,-69.584,-176.305,7.183,148.270
C01771=1216.673,317.208,-69.554,-176.307,7.180,148.269
C01772=1216.678,316.960,-69.523,-176.309,7.177,148.269
C01773=1216.682,316.712,-69.493,-176.312,7.175,148.269
C01774=1216.686,316.464,-69.463,-176.314,7.172,148.269
C01775=1216.691,316.216,-69.432,-176.316,7.170,148.270
C01776=1216.694,315.968,-69.402,-176.319,7.166,148.269
C01777=1216.699,315.720,-69.371,-176.321,7.164,148.269
C01778=1216.704,315.443,-69.337,-176.323,7.161,148.269
C01779=1216.708,315.168,-69.303,-176.326,7.158,148.269
C01780=1216.713,314.891,-69.270,-176.329,7.155,148.269
C01781=1216.718,314.616,-69.236,-176.331,7.153,148.269
C01782=1216.722,314.367,-69.206,-176.333,7.150,148.269
C01783=1216.727,314.119,-69.175,-176.336,7.148,148.269
C01784=1216.730,313.872,-69.145,-176.338,7.144,148.269
C01785=1216.735,313.623,-69.115,-176.340,7.142,148.269
C01786=1216.739,313.375,-69.085,-176.343,7.139,148.269
C01787=1216.743,313.127,-69.054,-176.345,7.137,148.269
C01788=1216.747,312.879,-69.024,-176.347,7.134,148.269
C01789=1216.752,312.631,-68.994,-176.349,7.132,148.269
C01790=1216.756,312.382,-68.964,-176.352,7.128,148.269
C01791=1216.761,312.134,-68.933,-176.354,7.126,148.269
C01792=1216.765,311.887,-68.903,-176.356,7.123,148.269
C01793=1216.770,311.638,-68.873,-176.359,7.121,148.269
C01794=1216.774,311.390,-68.843,-176.361,7.118,148.269
C01795=1216.778,311.142,-68.814,-176.363,7.115,148.269
C01796=1216.782,310.894,-68.783,-176.365,7.113,148.269
C01797=1216.786,310.645,-68.753,-176.368,7.110,148.269
C01798=1216.791,310.397,-68.722,-176.370,7.108,148.269
C01799=1216.795,310.149,-68.693,-176.373,7.105,148.269
C01800=1216.799,309.901,-68.662,-176.375,7.103,148.270
C01801=1216.804,309.653,-68.633,-176.377,7.099,148.269
C01802=1216.807,309.405,-68.602,-176.379,7.097,148.269
C01803=1216.812,309.157,-68.572,-176.382,7.094,148.269
C01804=1216.817,308.908,-68.543,-176.384,7.092,148.269
C01805=1216.820,308.661,-68.513,-176.387,7.089,148.269
C01806=1216.825,308.412,-68.483,-176.389,7.087,148.269
C01807=1216.829,308.164,-68.453,-176.391,7.084,148.270
C01808=1216.833,307.916,-68.423,-176.394,7.081,148.270
C01809=1216.838,307.668,-68.393,-176.396,7.079,148.270
C01810=1216.842,307.420,-68.363,-176.398,7.076,148.270
C01811=1216.846,307.172,-68.333,-176.401,7.074,148.270
